    movel([0.226532, -1.331171, -2.606399, -0.774819, 1.570796, 1.797328],accel_mss,speed_ms,0,blend_radius_m)
    movel([0.225717, -1.333588, -2.604857, -0.773944, 1.570796, 1.796514],accel_mss,speed_ms,0,blend_radius_m)
    movel([0.224908, -1.335996, -2.603314, -0.773080, 1.570796, 1.795704],accel_mss,speed_ms,0,blend_radius_m)
    movel([0.224102, -1.338394, -2.601768, -0.772227, 1.570796, 1.794898],accel_mss,speed_ms,0,blend_radius_m)
    movel([0.223301, -1.340783, -2.600221, -0.771385, 1.570796, 1.794097],accel_mss,speed_ms,0,blend_radius_m)
    movel([0.222504, -1.343162, -2.598672, -0.770555, 1.570796, 1.793300],accel_mss,speed_ms,0,blend_radius_m)
    movel([0.221711, -1.345532, -2.597121, -0.769735, 1.570796, 1.792507],accel_mss,speed_ms,0,blend_radius_m)
    movel([0.220923, -1.347893, -2.595569, -0.768927, 1.570796, 1.791719],accel_mss,speed_ms,0,blend_radius_m)
    movel([0.220138, -1.350245, -2.594015, -0.768129, 1.570796, 1.790935],accel_mss,speed_ms,0,blend_radius_m)
    movel([0.219358, -1.352588, -2.592459, -0.767341, 1.570796, 1.790154],accel_mss,speed_ms,0,blend_radius_m)
    movel([0.218582, -1.354923, -2.590901, -0.766565, 1.570796, 1.789378],accel_mss,speed_ms,0,blend_radius_m)
    movel([0.217810, -1.357248, -2.589342, -0.765799, 1.570796, 1.788606],accel_mss,speed_ms,0,blend_radius_m)
    movel([0.217042, -1.359565, -2.587781, -0.765043, 1.570796, 1.787838],accel_mss,speed_ms,0,blend_radius_m)
    movel([0.216277, -1.361873, -2.586219, -0.764298, 1.570796, 1.787074],accel_mss,speed_ms,0,blend_radius_m)
    movel([0.215517, -1.364172, -2.584655, -0.763562, 1.570796, 1.786314],accel_mss,speed_ms,0,blend_radius_m)
    movel([0.214761, -1.366463, -2.583089, -0.762837, 1.570796, 1.785557],accel_mss,speed_ms,0,blend_radius_m)
    # Splitting Linear movement in 4 (instruction 613: MoveL 496)
    movel([0.212425, -1.366695, -2.582929, -0.762764, 1.570796, 1.783222],accel_mss,speed_ms,0,blend_radius_m)
    movel([0.210088, -1.366933, -2.582767, -0.762689, 1.570796, 1.780884],accel_mss,speed_ms,0,blend_radius_m)
    movel([0.207750, -1.367175, -2.582601, -0.762613, 1.570796, 1.778546],accel_mss,speed_ms,0,blend_radius_m)
    movel([0.205411, -1.367422, -2.582431, -0.762536, 1.570796, 1.776207],accel_mss,speed_ms,0,blend_radius_m)
    speed_ms = 0.003
    # Splitting Linear movement in 8 (instruction 615: MoveL 497)
    movel([0.205411, -1.365756, -2.581675, -0.764958, 1.570796, 1.776207],accel_mss,speed_ms,0,blend_radius_m)
    movel([0.205411, -1.364096, -2.580917, -0.767376, 1.570796, 1.776207],accel_mss,speed_ms,0,blend_radius_m)
    movel([0.205411, -1.362442, -2.580157, -0.769790, 1.570796, 1.776207],accel_mss,speed_ms,0,blend_radius_m)
    movel([0.205411, -1.360794, -2.579395, -0.772200, 1.570796, 1.776207],accel_mss,speed_ms,0,blend_radius_m)
    movel([0.205411, -1.359151, -2.578631, -0.774607, 1.570796, 1.776207],accel_mss,speed_ms,0,blend_radius_m)
    movel([0.205411, -1.357515, -2.577864, -0.777010, 1.570796, 1.776207],accel_mss,speed_ms,0,blend_radius_m)
    movel([0.205411, -1.355884, -2.577096, -0.779409, 1.570796, 1.776207],accel_mss,speed_ms,0,blend_radius_m)
    movel([0.205411, -1.354259, -2.576326, -0.781804, 1.570796, 1.776207],accel_mss,speed_ms,0,blend_radius_m)
    speed_ms = 1.000
    # Splitting Linear movement in 12 (instruction 617: MoveL 498)
    movel([0.205411, -1.352102, -2.575295, -0.784992, 1.570796, 1.776207],accel_mss,speed_ms,0,blend_radius_m)
    movel([0.205411, -1.349954, -2.574261, -0.788174, 1.570796, 1.776207],accel_mss,speed_ms,0,blend_radius_m)
    movel([0.205411, -1.347818, -2.573223, -0.791348, 1.570796, 1.776207],accel_mss,speed_ms,0,blend_radius_m)
    movel([0.205411, -1.345691, -2.572182, -0.794516, 1.570796, 1.776207],accel_mss,speed_ms,0,blend_radius_m)
    movel([0.205411, -1.343575, -2.571137, -0.797677, 1.570796, 1.776207],accel_mss,speed_ms,0,blend_radius_m)
    movel([0.205411, -1.341469, -2.570088, -0.800832, 1.570796, 1.776207],accel_mss,speed_ms,0,blend_radius_m)
    movel([0.205411, -1.339373, -2.569036, -0.803980, 1.570796, 1.776207],accel_mss,speed_ms,0,blend_radius_m)
    movel([0.205411, -1.337288, -2.567980, -0.807121, 1.570796, 1.776207],accel_mss,speed_ms,0,blend_radius_m)
    movel([0.205411, -1.335213, -2.566921, -0.810255, 1.570796, 1.776207],accel_mss,speed_ms,0,blend_radius_m)
    movel([0.205411, -1.333148, -2.565858, -0.813383, 1.570796, 1.776207],accel_mss,speed_ms,0,blend_radius_m)
    movel([0.205411, -1.331093, -2.564792, -0.816504, 1.570796, 1.776207],accel_mss,speed_ms,0,blend_radius_m)
    movel([0.205411, -1.329048, -2.563722, -0.819619, 1.570796, 1.776207],accel_mss,speed_ms,0,blend_radius_m)
    # Splitting Linear movement in 4 (instruction 618: MoveL 499)
    movel([0.207507, -1.328481, -2.564090, -0.819818, 1.570796, 1.778304],accel_mss,speed_ms,0,blend_radius_m)
    movel([0.209605, -1.327917, -2.564455, -0.820017, 1.570796, 1.780401],accel_mss,speed_ms,0,blend_radius_m)
    movel([0.211703, -1.327356, -2.564818, -0.820215, 1.570796, 1.782499],accel_mss,speed_ms,0,blend_radius_m)
    movel([0.213802, -1.326799, -2.565178, -0.820412, 1.570796, 1.784598],accel_mss,speed_ms,0,blend_radius_m)
    # Splitting Linear movement in 12 (instruction 619: MoveL 500)
    movel([0.213802, -1.328846, -2.566251, -0.817292, 1.570796, 1.784598],accel_mss,speed_ms,0,blend_radius_m)
    movel([0.213802, -1.330904, -2.567319, -0.814166, 1.570796, 1.784598],accel_mss,speed_ms,0,blend_radius_m)
    movel([0.213802, -1.332972, -2.568384, -0.811033, 1.570796, 1.784598],accel_mss,speed_ms,0,blend_radius_m)
    movel([0.213802, -1.335050, -2.569446, -0.807893, 1.570796, 1.784598],accel_mss,speed_ms,0,blend_radius_m)
    movel([0.213802, -1.337139, -2.570504, -0.804746, 1.570796, 1.784598],accel_mss,speed_ms,0,blend_radius_m)
    movel([0.213802, -1.339237, -2.571559, -0.801593, 1.570796, 1.784598],accel_mss,speed_ms,0,blend_radius_m)
    movel([0.213802, -1.341346, -2.572610, -0.798433, 1.570796, 1.784598],accel_mss,speed_ms,0,blend_radius_m)
    movel([0.213802, -1.343466, -2.573657, -0.795266, 1.570796, 1.784598],accel_mss,speed_ms,0,blend_radius_m)
    movel([0.213802, -1.345596, -2.574701, -0.792092, 1.570796, 1.784598],accel_mss,speed_ms,0,blend_radius_m)
    movel([0.213802, -1.347736, -2.575741, -0.788912, 1.570796, 1.784598],accel_mss,speed_ms,0,blend_radius_m)
    movel([0.213802, -1.349887, -2.576778, -0.785725, 1.570796, 1.784598],accel_mss,speed_ms,0,blend_radius_m)
    movel([0.213802, -1.352047, -2.577811, -0.782531, 1.570796, 1.784598],accel_mss,speed_ms,0,blend_radius_m)
    speed_ms = 0.003
    # Splitting Linear movement in 6 (instruction 621: MoveL 501)
    movel([0.213802, -1.353675, -2.578583, -0.780131, 1.570796, 1.784598],accel_mss,speed_ms,0,blend_radius_m)
    movel([0.213802, -1.355308, -2.579353, -0.777727, 1.570796, 1.784598],accel_mss,speed_ms,0,blend_radius_m)
    movel([0.213802, -1.356948, -2.580121, -0.775320, 1.570796, 1.784598],accel_mss,speed_ms,0,blend_radius_m)
    movel([0.213802, -1.358593, -2.580887, -0.772909, 1.570796, 1.784598],accel_mss,speed_ms,0,blend_radius_m)
    movel([0.213802, -1.360244, -2.581651, -0.770494, 1.570796, 1.784598],accel_mss,speed_ms,0,blend_radius_m)
    movel([0.213802, -1.361901, -2.582413, -0.768075, 1.570796, 1.784598],accel_mss,speed_ms,0,blend_radius_m)
    speed_ms = 0.007
    # Splitting Linear movement in 28 (instruction 623: MoveL 502)
    movel([0.214539, -1.359700, -2.583906, -0.768782, 1.570796, 1.785335],accel_mss,speed_ms,0,blend_radius_m)
    movel([0.215280, -1.357492, -2.585397, -0.769499, 1.570796, 1.786076],accel_mss,speed_ms,0,blend_radius_m)
    movel([0.216024, -1.355276, -2.586887, -0.770226, 1.570796, 1.786820],accel_mss,speed_ms,0,blend_radius_m)
    movel([0.216772, -1.353052, -2.588375, -0.770962, 1.570796, 1.787569],accel_mss,speed_ms,0,blend_radius_m)
    movel([0.217524, -1.350820, -2.589862, -0.771707, 1.570796, 1.788321],accel_mss,speed_ms,0,blend_radius_m)
    movel([0.218280, -1.348579, -2.591347, -0.772462, 1.570796, 1.789076],accel_mss,speed_ms,0,blend_radius_m)
    movel([0.219040, -1.346331, -2.592831, -0.773227, 1.570796, 1.789836],accel_mss,speed_ms,0,blend_radius_m)
    movel([0.219803, -1.344074, -2.594313, -0.774002, 1.570796, 1.790599],accel_mss,speed_ms,0,blend_radius_m)
    movel([0.220570, -1.341809, -2.595793, -0.774786, 1.570796, 1.791367],accel_mss,speed_ms,0,blend_radius_m)
    movel([0.221341, -1.339536, -2.597272, -0.775581, 1.570796, 1.792138],accel_mss,speed_ms,0,blend_radius_m)
    movel([0.222116, -1.337254, -2.598749, -0.776385, 1.570796, 1.792913],accel_mss,speed_ms,0,blend_radius_m)
    movel([0.222895, -1.334964, -2.600225, -0.777200, 1.570796, 1.793692],accel_mss,speed_ms,0,blend_radius_m)
    movel([0.223679, -1.332665, -2.601699, -0.778024, 1.570796, 1.794475],accel_mss,speed_ms,0,blend_radius_m)
    movel([0.224466, -1.330358, -2.603171, -0.778860, 1.570796, 1.795262],accel_mss,speed_ms,0,blend_radius_m)
    movel([0.225257, -1.328042, -2.604642, -0.779705, 1.570796, 1.796053],accel_mss,speed_ms,0,blend_radius_m)
    movel([0.226052, -1.325717, -2.606111, -0.780561, 1.570796, 1.796848],accel_mss,speed_ms,0,blend_radius_m)
    movel([0.226851, -1.323383, -2.607578, -0.781427, 1.570796, 1.797648],accel_mss,speed_ms,0,blend_radius_m)
    movel([0.227655, -1.321040, -2.609044, -0.782305, 1.570796, 1.798451],accel_mss,speed_ms,0,blend_radius_m)
    movel([0.228462, -1.318689, -2.610508, -0.783192, 1.570796, 1.799259],accel_mss,speed_ms,0,blend_radius_m)
    movel([0.229274, -1.316328, -2.611970, -0.784091, 1.570796, 1.800071],accel_mss,speed_ms,0,blend_radius_m)
    movel([0.230091, -1.313958, -2.613431, -0.785001, 1.570796, 1.800887],accel_mss,speed_ms,0,blend_radius_m)
    movel([0.230911, -1.311578, -2.614889, -0.785921, 1.570796, 1.801707],accel_mss,speed_ms,0,blend_radius_m)
    movel([0.231736, -1.309190, -2.616346, -0.786853, 1.570796, 1.802532],accel_mss,speed_ms,0,blend_radius_m)
    movel([0.232565, -1.306792, -2.617802, -0.787796, 1.570796, 1.803361],accel_mss,speed_ms,0,blend_radius_m)
    movel([0.233399, -1.304384, -2.619255, -0.788750, 1.570796, 1.804195],accel_mss,speed_ms,0,blend_radius_m)
    movel([0.234237, -1.301967, -2.620707, -0.789716, 1.570796, 1.805033],accel_mss,speed_ms,0,blend_radius_m)
    movel([0.235079, -1.299540, -2.622156, -0.790693, 1.570796, 1.805875],accel_mss,speed_ms,0,blend_radius_m)
    movel([0.235926, -1.297103, -2.623604, -0.791681, 1.570796, 1.806722],accel_mss,speed_ms,0,blend_radius_m)
    # Splitting Linear movement in 6 (instruction 624: MoveC 503)
    movel([0.238136, -1.297220, -2.623535, -0.791634, 1.570796, 1.808932],accel_mss,speed_ms,0,blend_radius_m)
    movel([0.240342, -1.297342, -2.623463, -0.791584, 1.570796, 1.811138],accel_mss,speed_ms,0,blend_radius_m)
    movel([0.242546, -1.297469, -2.623388, -0.791532, 1.570796, 1.813342],accel_mss,speed_ms,0,blend_radius_m)
    movel([0.244746, -1.297602, -2.623309, -0.791478, 1.570796, 1.815543],accel_mss,speed_ms,0,blend_radius_m)
    movel([0.246944, -1.297740, -2.623227, -0.791422, 1.570796, 1.817740],accel_mss,speed_ms,0,blend_radius_m)
    movel([0.249138, -1.297883, -2.623142, -0.791364, 1.570796, 1.819935],accel_mss,speed_ms,0,blend_radius_m)
    # Splitting Linear movement in 12 (instruction 625: MoveC 504)
    movel([0.250068, -1.299641, -2.622096, -0.790652, 1.570796, 1.820865],accel_mss,speed_ms,0,blend_radius_m)
    movel([0.250994, -1.301398, -2.621047, -0.789944, 1.570796, 1.821791],accel_mss,speed_ms,0,blend_radius_m)
    movel([0.251916, -1.303152, -2.619996, -0.789241, 1.570796, 1.822712],accel_mss,speed_ms,0,blend_radius_m)
    movel([0.252833, -1.304905, -2.618941, -0.788543, 1.570796, 1.823629],accel_mss,speed_ms,0,blend_radius_m)
    movel([0.253746, -1.306655, -2.617884, -0.787850, 1.570796, 1.824542],accel_mss,speed_ms,0,blend_radius_m)
    movel([0.254655, -1.308403, -2.616824, -0.787161, 1.570796, 1.825451],accel_mss,speed_ms,0,blend_radius_m)
    movel([0.255560, -1.310150, -2.615762, -0.786478, 1.570796, 1.826356],accel_mss,speed_ms,0,blend_radius_m)
    movel([0.256461, -1.311894, -2.614696, -0.785799, 1.570796, 1.827257],accel_mss,speed_ms,0,blend_radius_m)
    movel([0.257357, -1.313636, -2.613628, -0.785125, 1.570796, 1.828154],accel_mss,speed_ms,0,blend_radius_m)
    movel([0.258250, -1.315377, -2.612557, -0.784455, 1.570796, 1.829046],accel_mss,speed_ms,0,blend_radius_m)
    movel([0.259138, -1.317115, -2.611484, -0.783791, 1.570796, 1.829934],accel_mss,speed_ms,0,blend_radius_m)
    movel([0.260023, -1.318851, -2.610407, -0.783131, 1.570796, 1.830819],accel_mss,speed_ms,0,blend_radius_m)
    movel([0.259481, -1.321910, -2.608501, -0.781978, 1.570796, 1.830277],accel_mss,speed_ms,0,blend_radius_m)
    movel([0.259060, -1.323596, -2.607445, -0.781348, 1.570796, 1.829856],accel_mss,speed_ms,0,blend_radius_m)
    movel([0.258139, -1.326541, -2.605592, -0.780257, 1.570796, 1.828935],accel_mss,speed_ms,0,blend_radius_m)
    movel([0.256608, -1.330373, -2.603162, -0.778854, 1.570796, 1.827405],accel_mss,speed_ms,0,blend_radius_m)
    movel([0.255647, -1.332392, -2.601874, -0.778123, 1.570796, 1.826443],accel_mss,speed_ms,0,blend_radius_m)
    movel([0.254869, -1.333870, -2.600928, -0.777592, 1.570796, 1.825665],accel_mss,speed_ms,0,blend_radius_m)
    # Splitting Linear movement in 8 (instruction 632: MoveC 511)
    movel([0.253270, -1.335839, -2.599662, -0.776888, 1.570796, 1.824066],accel_mss,speed_ms,0,blend_radius_m)
    movel([0.251678, -1.337802, -2.598395, -0.776191, 1.570796, 1.822474],accel_mss,speed_ms,0,blend_radius_m)
    movel([0.250091, -1.339760, -2.597127, -0.775502, 1.570796, 1.820888],accel_mss,speed_ms,0,blend_radius_m)
    movel([0.248511, -1.341712, -2.595857, -0.774820, 1.570796, 1.819308],accel_mss,speed_ms,0,blend_radius_m)
    movel([0.246938, -1.343658, -2.594586, -0.774145, 1.570796, 1.817734],accel_mss,speed_ms,0,blend_radius_m)
    movel([0.245370, -1.345598, -2.593313, -0.773478, 1.570796, 1.816166],accel_mss,speed_ms,0,blend_radius_m)
    movel([0.243809, -1.347533, -2.592038, -0.772817, 1.570796, 1.814605],accel_mss,speed_ms,0,blend_radius_m)
    movel([0.242253, -1.349462, -2.590763, -0.772164, 1.570796, 1.813050],accel_mss,speed_ms,0,blend_radius_m)
    # Splitting Linear movement in 4 (instruction 633: MoveC 512)
    movel([0.240979, -1.350466, -2.590097, -0.771826, 1.570796, 1.811775],accel_mss,speed_ms,0,blend_radius_m)
    movel([0.239707, -1.351470, -2.589430, -0.771489, 1.570796, 1.810503],accel_mss,speed_ms,0,blend_radius_m)
    movel([0.238437, -1.352472, -2.588763, -0.771155, 1.570796, 1.809234],accel_mss,speed_ms,0,blend_radius_m)
    movel([0.237170, -1.353473, -2.588094, -0.770822, 1.570796, 1.807966],accel_mss,speed_ms,0,blend_radius_m)
    movel([0.235144, -1.354822, -2.587191, -0.770375, 1.570796, 1.805940],accel_mss,speed_ms,0,blend_radius_m)
    # Splitting Linear movement in 8 (instruction 635: MoveC 514)
    movel([0.233110, -1.355638, -2.586644, -0.770107, 1.570796, 1.803906],accel_mss,speed_ms,0,blend_radius_m)
    movel([0.231078, -1.356455, -2.586095, -0.769838, 1.570796, 1.801874],accel_mss,speed_ms,0,blend_radius_m)
    movel([0.229048, -1.357274, -2.585544, -0.769571, 1.570796, 1.799845],accel_mss,speed_ms,0,blend_radius_m)
    movel([0.227021, -1.358095, -2.584991, -0.769303, 1.570796, 1.797817],accel_mss,speed_ms,0,blend_radius_m)
    movel([0.224995, -1.358917, -2.584436, -0.769036, 1.570796, 1.795791],accel_mss,speed_ms,0,blend_radius_m)
    movel([0.222972, -1.359741, -2.583878, -0.768769, 1.570796, 1.793768],accel_mss,speed_ms,0,blend_radius_m)
    movel([0.220950, -1.360567, -2.583319, -0.768503, 1.570796, 1.791747],accel_mss,speed_ms,0,blend_radius_m)
    movel([0.218931, -1.361394, -2.582758, -0.768237, 1.570796, 1.789728],accel_mss,speed_ms,0,blend_radius_m)
    # Splitting Linear movement in 4 (instruction 636: MoveC 515)
    movel([0.217650, -1.361519, -2.582673, -0.768197, 1.570796, 1.788446],accel_mss,speed_ms,0,blend_radius_m)
    movel([0.216367, -1.361645, -2.582587, -0.768157, 1.570796, 1.787164],accel_mss,speed_ms,0,blend_radius_m)
    movel([0.215085, -1.361772, -2.582501, -0.768116, 1.570796, 1.785881],accel_mss,speed_ms,0,blend_radius_m)
    movel([0.213802, -1.361901, -2.582413, -0.768075, 1.570796, 1.784598],accel_mss,speed_ms,0,blend_radius_m)
    speed_ms = 0.003
    movel([0.213802, -1.365233, -2.583931, -0.763226, 1.570796, 1.784598],accel_mss,speed_ms,0,blend_radius_m)
    speed_ms = 0.007
    # Splitting Linear movement in 28 (instruction 640: MoveL 517)
    movel([0.214539, -1.363038, -2.585427, -0.763924, 1.570796, 1.785335],accel_mss,speed_ms,0,blend_radius_m)
    movel([0.215280, -1.360835, -2.586922, -0.764632, 1.570796, 1.786076],accel_mss,speed_ms,0,blend_radius_m)
    movel([0.216024, -1.358625, -2.588416, -0.765349, 1.570796, 1.786820],accel_mss,speed_ms,0,blend_radius_m)
    movel([0.216772, -1.356406, -2.589908, -0.766075, 1.570796, 1.787569],accel_mss,speed_ms,0,blend_radius_m)
    movel([0.217524, -1.354180, -2.591398, -0.766811, 1.570796, 1.788321],accel_mss,speed_ms,0,blend_radius_m)
    movel([0.218280, -1.351945, -2.592887, -0.767557, 1.570796, 1.789076],accel_mss,speed_ms,0,blend_radius_m)
    movel([0.219040, -1.349703, -2.594374, -0.768312, 1.570796, 1.789836],accel_mss,speed_ms,0,blend_radius_m)
    movel([0.219803, -1.347452, -2.595860, -0.769077, 1.570796, 1.790599],accel_mss,speed_ms,0,blend_radius_m)
    movel([0.220570, -1.345192, -2.597344, -0.769852, 1.570796, 1.791367],accel_mss,speed_ms,0,blend_radius_m)
    movel([0.221341, -1.342925, -2.598827, -0.770637, 1.570796, 1.792138],accel_mss,speed_ms,0,blend_radius_m)
    movel([0.222116, -1.340649, -2.600308, -0.771432, 1.570796, 1.792913],accel_mss,speed_ms,0,blend_radius_m)
    movel([0.222895, -1.338364, -2.601787, -0.772237, 1.570796, 1.793692],accel_mss,speed_ms,0,blend_radius_m)
    movel([0.223679, -1.336071, -2.603265, -0.773053, 1.570796, 1.794475],accel_mss,speed_ms,0,blend_radius_m)
    movel([0.224466, -1.333769, -2.604741, -0.773878, 1.570796, 1.795262],accel_mss,speed_ms,0,blend_radius_m)
    movel([0.225257, -1.331459, -2.606216, -0.774714, 1.570796, 1.796053],accel_mss,speed_ms,0,blend_radius_m)
    movel([0.226052, -1.329140, -2.607689, -0.775561, 1.570796, 1.796848],accel_mss,speed_ms,0,blend_radius_m)
    movel([0.226851, -1.326811, -2.609160, -0.776418, 1.570796, 1.797648],accel_mss,speed_ms,0,blend_radius_m)
    movel([0.227655, -1.324474, -2.610630, -0.777285, 1.570796, 1.798451],accel_mss,speed_ms,0,blend_radius_m)
    movel([0.228462, -1.322128, -2.612098, -0.778163, 1.570796, 1.799259],accel_mss,speed_ms,0,blend_radius_m)
    movel([0.229274, -1.319773, -2.613564, -0.779053, 1.570796, 1.800071],accel_mss,speed_ms,0,blend_radius_m)
    movel([0.230091, -1.317408, -2.615028, -0.779953, 1.570796, 1.800887],accel_mss,speed_ms,0,blend_radius_m)
    movel([0.230911, -1.315034, -2.616491, -0.780864, 1.570796, 1.801707],accel_mss,speed_ms,0,blend_radius_m)
    movel([0.231736, -1.312651, -2.617952, -0.781786, 1.570796, 1.802532],accel_mss,speed_ms,0,blend_radius_m)
    movel([0.232565, -1.310259, -2.619411, -0.782719, 1.570796, 1.803361],accel_mss,speed_ms,0,blend_radius_m)
    movel([0.233399, -1.307857, -2.620869, -0.783664, 1.570796, 1.804195],accel_mss,speed_ms,0,blend_radius_m)
    movel([0.234237, -1.305445, -2.622325, -0.784620, 1.570796, 1.805033],accel_mss,speed_ms,0,blend_radius_m)
    movel([0.235079, -1.303023, -2.623778, -0.785587, 1.570796, 1.805875],accel_mss,speed_ms,0,blend_radius_m)
    movel([0.235926, -1.300592, -2.625231, -0.786566, 1.570796, 1.806722],accel_mss,speed_ms,0,blend_radius_m)
    # Splitting Linear movement in 6 (instruction 641: MoveC 518)
    movel([0.238136, -1.300709, -2.625161, -0.786519, 1.570796, 1.808932],accel_mss,speed_ms,0,blend_radius_m)
    movel([0.240342, -1.300830, -2.625089, -0.786470, 1.570796, 1.811138],accel_mss,speed_ms,0,blend_radius_m)
    movel([0.242546, -1.300957, -2.625013, -0.786419, 1.570796, 1.813342],accel_mss,speed_ms,0,blend_radius_m)
    movel([0.244746, -1.301090, -2.624934, -0.786365, 1.570796, 1.815543],accel_mss,speed_ms,0,blend_radius_m)
    movel([0.246944, -1.301227, -2.624852, -0.786310, 1.570796, 1.817740],accel_mss,speed_ms,0,blend_radius_m)
    movel([0.249138, -1.301370, -2.624767, -0.786252, 1.570796, 1.819935],accel_mss,speed_ms,0,blend_radius_m)
    # Splitting Linear movement in 12 (instruction 642: MoveC 519)
    movel([0.250068, -1.303125, -2.623718, -0.785547, 1.570796, 1.820865],accel_mss,speed_ms,0,blend_radius_m)
    movel([0.250994, -1.304877, -2.622666, -0.784846, 1.570796, 1.821791],accel_mss,speed_ms,0,blend_radius_m)
    movel([0.251916, -1.306628, -2.621612, -0.784150, 1.570796, 1.822712],accel_mss,speed_ms,0,blend_radius_m)
    movel([0.252833, -1.308376, -2.620554, -0.783459, 1.570796, 1.823629],accel_mss,speed_ms,0,blend_radius_m)
    movel([0.253746, -1.310122, -2.619494, -0.782772, 1.570796, 1.824542],accel_mss,speed_ms,0,blend_radius_m)
    movel([0.254655, -1.311867, -2.618431, -0.782091, 1.570796, 1.825451],accel_mss,speed_ms,0,blend_radius_m)
    movel([0.255560, -1.313609, -2.617366, -0.781414, 1.570796, 1.826356],accel_mss,speed_ms,0,blend_radius_m)
    movel([0.256461, -1.315349, -2.616297, -0.780742, 1.570796, 1.827257],accel_mss,speed_ms,0,blend_radius_m)
    movel([0.257357, -1.317088, -2.615226, -0.780075, 1.570796, 1.828154],accel_mss,speed_ms,0,blend_radius_m)
    movel([0.258250, -1.318824, -2.614152, -0.779413, 1.570796, 1.829046],accel_mss,speed_ms,0,blend_radius_m)
    movel([0.259138, -1.320558, -2.613076, -0.778755, 1.570796, 1.829934],accel_mss,speed_ms,0,blend_radius_m)
    movel([0.260023, -1.322290, -2.611997, -0.778103, 1.570796, 1.830819],accel_mss,speed_ms,0,blend_radius_m)
    movel([0.259481, -1.325342, -2.610085, -0.776962, 1.570796, 1.830277],accel_mss,speed_ms,0,blend_radius_m)
    movel([0.259060, -1.327024, -2.609026, -0.776339, 1.570796, 1.829856],accel_mss,speed_ms,0,blend_radius_m)
    movel([0.258139, -1.329961, -2.607168, -0.775260, 1.570796, 1.828935],accel_mss,speed_ms,0,blend_radius_m)
    movel([0.256608, -1.333784, -2.604732, -0.773873, 1.570796, 1.827405],accel_mss,speed_ms,0,blend_radius_m)
    movel([0.255647, -1.335798, -2.603441, -0.773150, 1.570796, 1.826443],accel_mss,speed_ms,0,blend_radius_m)
    movel([0.254869, -1.337272, -2.602492, -0.772625, 1.570796, 1.825665],accel_mss,speed_ms,0,blend_radius_m)
    # Splitting Linear movement in 8 (instruction 649: MoveC 526)
    movel([0.253270, -1.339237, -2.601223, -0.771929, 1.570796, 1.824066],accel_mss,speed_ms,0,blend_radius_m)
    movel([0.251678, -1.341195, -2.599953, -0.771241, 1.570796, 1.822474],accel_mss,speed_ms,0,blend_radius_m)
    movel([0.250091, -1.343148, -2.598681, -0.770560, 1.570796, 1.820888],accel_mss,speed_ms,0,blend_radius_m)
    movel([0.248511, -1.345095, -2.597408, -0.769886, 1.570796, 1.819308],accel_mss,speed_ms,0,blend_radius_m)
    movel([0.246938, -1.347036, -2.596133, -0.769219, 1.570796, 1.817734],accel_mss,speed_ms,0,blend_radius_m)
    movel([0.245370, -1.348972, -2.594857, -0.768560, 1.570796, 1.816166],accel_mss,speed_ms,0,blend_radius_m)
    movel([0.243809, -1.350902, -2.593580, -0.767907, 1.570796, 1.814605],accel_mss,speed_ms,0,blend_radius_m)
    movel([0.242253, -1.352826, -2.592301, -0.767262, 1.570796, 1.813050],accel_mss,speed_ms,0,blend_radius_m)
    # Splitting Linear movement in 4 (instruction 650: MoveC 527)
    movel([0.240979, -1.353828, -2.591633, -0.766928, 1.570796, 1.811775],accel_mss,speed_ms,0,blend_radius_m)
    movel([0.239707, -1.354828, -2.590965, -0.766596, 1.570796, 1.810503],accel_mss,speed_ms,0,blend_radius_m)
    movel([0.238437, -1.355828, -2.590296, -0.766266, 1.570796, 1.809234],accel_mss,speed_ms,0,blend_radius_m)
    movel([0.237170, -1.356826, -2.589626, -0.765937, 1.570796, 1.807966],accel_mss,speed_ms,0,blend_radius_m)
    movel([0.235144, -1.358172, -2.588720, -0.765496, 1.570796, 1.805940],accel_mss,speed_ms,0,blend_radius_m)
    # Splitting Linear movement in 8 (instruction 652: MoveC 529)
    movel([0.233110, -1.358986, -2.588172, -0.765231, 1.570796, 1.803906],accel_mss,speed_ms,0,blend_radius_m)
    movel([0.231078, -1.359801, -2.587622, -0.764966, 1.570796, 1.801874],accel_mss,speed_ms,0,blend_radius_m)
    movel([0.229048, -1.360618, -2.587069, -0.764702, 1.570796, 1.799845],accel_mss,speed_ms,0,blend_radius_m)
    movel([0.227021, -1.361436, -2.586515, -0.764438, 1.570796, 1.797817],accel_mss,speed_ms,0,blend_radius_m)
    movel([0.224995, -1.362257, -2.585958, -0.764174, 1.570796, 1.795791],accel_mss,speed_ms,0,blend_radius_m)
    movel([0.222972, -1.363079, -2.585399, -0.763911, 1.570796, 1.793768],accel_mss,speed_ms,0,blend_radius_m)
    movel([0.220950, -1.363902, -2.584839, -0.763648, 1.570796, 1.791747],accel_mss,speed_ms,0,blend_radius_m)
    movel([0.218931, -1.364727, -2.584276, -0.763386, 1.570796, 1.789728],accel_mss,speed_ms,0,blend_radius_m)
    # Splitting Linear movement in 4 (instruction 653: MoveC 530)
    movel([0.217650, -1.364851, -2.584191, -0.763347, 1.570796, 1.788446],accel_mss,speed_ms,0,blend_radius_m)
    movel([0.216367, -1.364977, -2.584105, -0.763307, 1.570796, 1.787164],accel_mss,speed_ms,0,blend_radius_m)
    movel([0.215085, -1.365104, -2.584018, -0.763266, 1.570796, 1.785881],accel_mss,speed_ms,0,blend_radius_m)
    movel([0.213802, -1.365233, -2.583931, -0.763226, 1.570796, 1.784598],accel_mss,speed_ms,0,blend_radius_m)
    speed_ms = 0.003
    # Splitting Linear movement in 6 (instruction 655: MoveL 531)
    movel([0.213802, -1.363009, -2.582920, -0.766460, 1.570796, 1.784598],accel_mss,speed_ms,0,blend_radius_m)
    movel([0.213802, -1.360796, -2.581906, -0.769688, 1.570796, 1.784598],accel_mss,speed_ms,0,blend_radius_m)
    movel([0.213802, -1.358593, -2.580887, -0.772909, 1.570796, 1.784598],accel_mss,speed_ms,0,blend_radius_m)
    movel([0.213802, -1.356401, -2.579865, -0.776123, 1.570796, 1.784598],accel_mss,speed_ms,0,blend_radius_m)
    movel([0.213802, -1.354219, -2.578840, -0.779330, 1.570796, 1.784598],accel_mss,speed_ms,0,blend_radius_m)
    movel([0.213802, -1.352047, -2.577811, -0.782531, 1.570796, 1.784598],accel_mss,speed_ms,0,blend_radius_m)
    speed_ms = 1.000
    # Splitting Linear movement in 12 (instruction 657: MoveL 532)
    movel([0.213802, -1.349887, -2.576778, -0.785725, 1.570796, 1.784598],accel_mss,speed_ms,0,blend_radius_m)
    movel([0.213802, -1.347736, -2.575741, -0.788912, 1.570796, 1.784598],accel_mss,speed_ms,0,blend_radius_m)
    movel([0.213802, -1.345596, -2.574701, -0.792092, 1.570796, 1.784598],accel_mss,speed_ms,0,blend_radius_m)
    movel([0.213802, -1.343466, -2.573657, -0.795266, 1.570796, 1.784598],accel_mss,speed_ms,0,blend_radius_m)
    movel([0.213802, -1.341346, -2.572610, -0.798433, 1.570796, 1.784598],accel_mss,speed_ms,0,blend_radius_m)
    movel([0.213802, -1.339237, -2.571559, -0.801593, 1.570796, 1.784598],accel_mss,speed_ms,0,blend_radius_m)
    movel([0.213802, -1.337139, -2.570504, -0.804746, 1.570796, 1.784598],accel_mss,speed_ms,0,blend_radius_m)
    movel([0.213802, -1.335050, -2.569446, -0.807893, 1.570796, 1.784598],accel_mss,speed_ms,0,blend_radius_m)
    movel([0.213802, -1.332972, -2.568384, -0.811033, 1.570796, 1.784598],accel_mss,speed_ms,0,blend_radius_m)
    movel([0.213802, -1.330904, -2.567319, -0.814166, 1.570796, 1.784598],accel_mss,speed_ms,0,blend_radius_m)
    movel([0.213802, -1.328846, -2.566251, -0.817292, 1.570796, 1.784598],accel_mss,speed_ms,0,blend_radius_m)
    movel([0.213802, -1.326799, -2.565178, -0.820412, 1.570796, 1.784598],accel_mss,speed_ms,0,blend_radius_m)
    # Splitting Linear movement in 18 (instruction 658: MoveL 533)
    movel([0.215158, -1.324599, -2.566596, -0.821194, 1.570796, 1.785954],accel_mss,speed_ms,0,blend_radius_m)
    movel([0.216520, -1.322393, -2.568011, -0.821985, 1.570796, 1.787317],accel_mss,speed_ms,0,blend_radius_m)
    movel([0.217889, -1.320180, -2.569425, -0.822785, 1.570796, 1.788685],accel_mss,speed_ms,0,blend_radius_m)
    movel([0.219264, -1.317959, -2.570837, -0.823593, 1.570796, 1.790060],accel_mss,speed_ms,0,blend_radius_m)
    movel([0.220645, -1.315730, -2.572247, -0.824411, 1.570796, 1.791441],accel_mss,speed_ms,0,blend_radius_m)
    movel([0.222033, -1.313495, -2.573656, -0.825238, 1.570796, 1.792829],accel_mss,speed_ms,0,blend_radius_m)
    movel([0.223426, -1.311251, -2.575063, -0.826075, 1.570796, 1.794223],accel_mss,speed_ms,0,blend_radius_m)
    movel([0.224827, -1.309001, -2.576468, -0.826920, 1.570796, 1.795623],accel_mss,speed_ms,0,blend_radius_m)
    movel([0.226234, -1.306742, -2.577872, -0.827775, 1.570796, 1.797030],accel_mss,speed_ms,0,blend_radius_m)
    movel([0.227647, -1.304476, -2.579273, -0.828640, 1.570796, 1.798444],accel_mss,speed_ms,0,blend_radius_m)
    movel([0.229067, -1.302202, -2.580673, -0.829513, 1.570796, 1.799864],accel_mss,speed_ms,0,blend_radius_m)
    movel([0.230494, -1.299921, -2.582071, -0.830397, 1.570796, 1.801290],accel_mss,speed_ms,0,blend_radius_m)
    movel([0.231927, -1.297632, -2.583468, -0.831290, 1.570796, 1.802724],accel_mss,speed_ms,0,blend_radius_m)
    movel([0.233367, -1.295334, -2.584862, -0.832193, 1.570796, 1.804164],accel_mss,speed_ms,0,blend_radius_m)
    movel([0.234814, -1.293029, -2.586255, -0.833105, 1.570796, 1.805610],accel_mss,speed_ms,0,blend_radius_m)
    movel([0.236268, -1.290716, -2.587646, -0.834028, 1.570796, 1.807064],accel_mss,speed_ms,0,blend_radius_m)
    movel([0.237728, -1.288394, -2.589035, -0.834960, 1.570796, 1.808525],accel_mss,speed_ms,0,blend_radius_m)
    movel([0.239196, -1.286065, -2.590422, -0.835902, 1.570796, 1.809992],accel_mss,speed_ms,0,blend_radius_m)
    # Splitting Linear movement in 12 (instruction 659: MoveL 534)
    movel([0.239196, -1.288161, -2.591538, -0.832691, 1.570796, 1.809992],accel_mss,speed_ms,0,blend_radius_m)
    movel([0.239196, -1.290267, -2.592650, -0.829471, 1.570796, 1.809992],accel_mss,speed_ms,0,blend_radius_m)
    movel([0.239196, -1.292386, -2.593759, -0.826244, 1.570796, 1.809992],accel_mss,speed_ms,0,blend_radius_m)
    movel([0.239196, -1.294515, -2.594865, -0.823009, 1.570796, 1.809992],accel_mss,speed_ms,0,blend_radius_m)
    movel([0.239196, -1.296656, -2.595967, -0.819766, 1.570796, 1.809992],accel_mss,speed_ms,0,blend_radius_m)
    movel([0.239196, -1.298808, -2.597065, -0.816516, 1.570796, 1.809992],accel_mss,speed_ms,0,blend_radius_m)
    movel([0.239196, -1.300972, -2.598160, -0.813257, 1.570796, 1.809992],accel_mss,speed_ms,0,blend_radius_m)
    movel([0.239196, -1.303147, -2.599252, -0.809991, 1.570796, 1.809992],accel_mss,speed_ms,0,blend_radius_m)
    movel([0.239196, -1.305333, -2.600340, -0.806716, 1.570796, 1.809992],accel_mss,speed_ms,0,blend_radius_m)
    movel([0.239196, -1.307531, -2.601424, -0.803434, 1.570796, 1.809992],accel_mss,speed_ms,0,blend_radius_m)
    movel([0.239196, -1.309740, -2.602505, -0.800144, 1.570796, 1.809992],accel_mss,speed_ms,0,blend_radius_m)
    movel([0.239196, -1.311961, -2.603582, -0.796846, 1.570796, 1.809992],accel_mss,speed_ms,0,blend_radius_m)
    speed_ms = 0.003
    # Splitting Linear movement in 6 (instruction 661: MoveL 535)
    movel([0.239196, -1.313634, -2.604387, -0.794368, 1.570796, 1.809992],accel_mss,speed_ms,0,blend_radius_m)
    movel([0.239196, -1.315314, -2.605191, -0.791884, 1.570796, 1.809992],accel_mss,speed_ms,0,blend_radius_m)
    movel([0.239196, -1.317000, -2.605992, -0.789397, 1.570796, 1.809992],accel_mss,speed_ms,0,blend_radius_m)
    movel([0.239196, -1.318693, -2.606791, -0.786905, 1.570796, 1.809992],accel_mss,speed_ms,0,blend_radius_m)
    movel([0.239196, -1.320392, -2.607588, -0.784409, 1.570796, 1.809992],accel_mss,speed_ms,0,blend_radius_m)
    movel([0.239196, -1.322098, -2.608383, -0.781908, 1.570796, 1.809992],accel_mss,speed_ms,0,blend_radius_m)
    speed_ms = 0.007
    # Splitting Linear movement in 4 (instruction 663: MoveC 536)
    movel([0.238117, -1.321461, -2.608781, -0.782146, 1.570796, 1.808913],accel_mss,speed_ms,0,blend_radius_m)
    movel([0.237036, -1.320826, -2.609178, -0.782385, 1.570796, 1.807833],accel_mss,speed_ms,0,blend_radius_m)
    movel([0.235953, -1.320192, -2.609573, -0.782624, 1.570796, 1.806750],accel_mss,speed_ms,0,blend_radius_m)
    movel([0.234868, -1.319559, -2.609967, -0.782863, 1.570796, 1.805664],accel_mss,speed_ms,0,blend_radius_m)
    movel([0.235037, -1.314955, -2.612817, -0.784617, 1.570796, 1.805833],accel_mss,speed_ms,0,blend_radius_m)
    # Splitting Linear movement in 4 (instruction 665: MoveC 538)
    movel([0.235966, -1.313583, -2.613661, -0.785145, 1.570796, 1.806762],accel_mss,speed_ms,0,blend_radius_m)
    movel([0.236897, -1.312208, -2.614504, -0.785677, 1.570796, 1.807694],accel_mss,speed_ms,0,blend_radius_m)
    movel([0.237832, -1.310830, -2.615347, -0.786212, 1.570796, 1.808628],accel_mss,speed_ms,0,blend_radius_m)
    movel([0.238769, -1.309448, -2.616189, -0.786752, 1.570796, 1.809565],accel_mss,speed_ms,0,blend_radius_m)
    # Splitting Linear movement in 4 (instruction 666: MoveC 539)
    movel([0.240367, -1.308658, -2.616670, -0.787061, 1.570796, 1.811164],accel_mss,speed_ms,0,blend_radius_m)
    movel([0.241968, -1.307867, -2.617150, -0.787372, 1.570796, 1.812764],accel_mss,speed_ms,0,blend_radius_m)
    movel([0.243570, -1.307078, -2.617628, -0.787683, 1.570796, 1.814366],accel_mss,speed_ms,0,blend_radius_m)
    movel([0.245174, -1.306289, -2.618106, -0.787995, 1.570796, 1.815970],accel_mss,speed_ms,0,blend_radius_m)
    movel([0.245654, -1.306259, -2.618124, -0.788006, 1.570796, 1.816450],accel_mss,speed_ms,0,blend_radius_m)
    # Splitting Linear movement in 4 (instruction 668: MoveC 541)
    movel([0.246742, -1.306911, -2.617729, -0.787749, 1.570796, 1.817539],accel_mss,speed_ms,0,blend_radius_m)
    movel([0.247828, -1.307565, -2.617333, -0.787491, 1.570796, 1.818625],accel_mss,speed_ms,0,blend_radius_m)
    movel([0.248912, -1.308220, -2.616936, -0.787233, 1.570796, 1.819708],accel_mss,speed_ms,0,blend_radius_m)
    movel([0.249994, -1.308876, -2.616537, -0.786976, 1.570796, 1.820790],accel_mss,speed_ms,0,blend_radius_m)
    movel([0.249744, -1.313555, -2.613678, -0.785156, 1.570796, 1.820541],accel_mss,speed_ms,0,blend_radius_m)
    # Splitting Linear movement in 4 (instruction 670: MoveC 543)
    movel([0.248800, -1.314923, -2.612837, -0.784629, 1.570796, 1.819596],accel_mss,speed_ms,0,blend_radius_m)
    movel([0.247858, -1.316287, -2.611996, -0.784107, 1.570796, 1.818654],accel_mss,speed_ms,0,blend_radius_m)
    movel([0.246918, -1.317648, -2.611154, -0.783588, 1.570796, 1.817715],accel_mss,speed_ms,0,blend_radius_m)
    movel([0.245982, -1.319006, -2.610311, -0.783072, 1.570796, 1.816778],accel_mss,speed_ms,0,blend_radius_m)
    # Splitting Linear movement in 4 (instruction 671: MoveC 544)
    movel([0.244401, -1.319771, -2.609835, -0.782783, 1.570796, 1.815197],accel_mss,speed_ms,0,blend_radius_m)
    movel([0.242822, -1.320536, -2.609358, -0.782494, 1.570796, 1.813618],accel_mss,speed_ms,0,blend_radius_m)
    movel([0.241244, -1.321303, -2.608880, -0.782206, 1.570796, 1.812040],accel_mss,speed_ms,0,blend_radius_m)
    movel([0.239668, -1.322069, -2.608401, -0.781918, 1.570796, 1.810464],accel_mss,speed_ms,0,blend_radius_m)
    movel([0.239196, -1.322098, -2.608383, -0.781908, 1.570796, 1.809992],accel_mss,speed_ms,0,blend_radius_m)
    speed_ms = 0.003
    movel([0.239196, -1.325529, -2.609967, -0.776893, 1.570796, 1.809992],accel_mss,speed_ms,0,blend_radius_m)
    speed_ms = 0.007
    # Splitting Linear movement in 4 (instruction 676: MoveC 547)
    movel([0.238117, -1.324894, -2.610366, -0.777129, 1.570796, 1.808913],accel_mss,speed_ms,0,blend_radius_m)
    movel([0.237036, -1.324260, -2.610764, -0.777365, 1.570796, 1.807833],accel_mss,speed_ms,0,blend_radius_m)
    movel([0.235953, -1.323628, -2.611160, -0.777601, 1.570796, 1.806750],accel_mss,speed_ms,0,blend_radius_m)
    movel([0.234868, -1.322997, -2.611555, -0.777837, 1.570796, 1.805664],accel_mss,speed_ms,0,blend_radius_m)
    movel([0.235037, -1.318403, -2.614413, -0.779573, 1.570796, 1.805833],accel_mss,speed_ms,0,blend_radius_m)
    # Splitting Linear movement in 4 (instruction 678: MoveC 549)
    movel([0.235966, -1.317034, -2.615259, -0.780096, 1.570796, 1.806762],accel_mss,speed_ms,0,blend_radius_m)
    movel([0.236897, -1.315662, -2.616105, -0.780622, 1.570796, 1.807694],accel_mss,speed_ms,0,blend_radius_m)
    movel([0.237832, -1.314287, -2.616950, -0.781152, 1.570796, 1.808628],accel_mss,speed_ms,0,blend_radius_m)
    movel([0.238769, -1.312909, -2.617794, -0.781686, 1.570796, 1.809565],accel_mss,speed_ms,0,blend_radius_m)
    # Splitting Linear movement in 4 (instruction 679: MoveC 550)
    movel([0.240367, -1.312120, -2.618276, -0.781992, 1.570796, 1.811164],accel_mss,speed_ms,0,blend_radius_m)
    movel([0.241968, -1.311332, -2.618758, -0.782299, 1.570796, 1.812764],accel_mss,speed_ms,0,blend_radius_m)
    movel([0.243570, -1.310544, -2.619238, -0.782607, 1.570796, 1.814366],accel_mss,speed_ms,0,blend_radius_m)
    movel([0.245174, -1.309757, -2.619716, -0.782916, 1.570796, 1.815970],accel_mss,speed_ms,0,blend_radius_m)
    movel([0.245654, -1.309727, -2.619735, -0.782928, 1.570796, 1.816450],accel_mss,speed_ms,0,blend_radius_m)
    # Splitting Linear movement in 4 (instruction 681: MoveC 552)
    movel([0.246742, -1.310378, -2.619339, -0.782672, 1.570796, 1.817539],accel_mss,speed_ms,0,blend_radius_m)
    movel([0.247828, -1.311030, -2.618942, -0.782417, 1.570796, 1.818625],accel_mss,speed_ms,0,blend_radius_m)
    movel([0.248912, -1.311684, -2.618543, -0.782162, 1.570796, 1.819708],accel_mss,speed_ms,0,blend_radius_m)
    movel([0.249994, -1.312338, -2.618143, -0.781907, 1.570796, 1.820790],accel_mss,speed_ms,0,blend_radius_m)
    movel([0.249744, -1.317007, -2.615276, -0.780106, 1.570796, 1.820541],accel_mss,speed_ms,0,blend_radius_m)
    # Splitting Linear movement in 4 (instruction 683: MoveC 554)
    movel([0.248800, -1.318371, -2.614433, -0.779585, 1.570796, 1.819596],accel_mss,speed_ms,0,blend_radius_m)
    movel([0.247858, -1.319732, -2.613589, -0.779068, 1.570796, 1.818654],accel_mss,speed_ms,0,blend_radius_m)
    movel([0.246918, -1.321090, -2.612745, -0.778555, 1.570796, 1.817715],accel_mss,speed_ms,0,blend_radius_m)
    movel([0.245982, -1.322444, -2.611900, -0.778045, 1.570796, 1.816778],accel_mss,speed_ms,0,blend_radius_m)
    # Splitting Linear movement in 4 (instruction 684: MoveC 555)
    movel([0.244401, -1.323208, -2.611423, -0.777758, 1.570796, 1.815197],accel_mss,speed_ms,0,blend_radius_m)
    movel([0.242822, -1.323971, -2.610945, -0.777473, 1.570796, 1.813618],accel_mss,speed_ms,0,blend_radius_m)
    movel([0.241244, -1.324736, -2.610466, -0.777188, 1.570796, 1.812040],accel_mss,speed_ms,0,blend_radius_m)
    movel([0.239668, -1.325501, -2.609985, -0.776903, 1.570796, 1.810464],accel_mss,speed_ms,0,blend_radius_m)
    movel([0.239196, -1.325529, -2.609967, -0.776893, 1.570796, 1.809992],accel_mss,speed_ms,0,blend_radius_m)
    speed_ms = 0.003
    # Splitting Linear movement in 6 (instruction 687: MoveL 557)
    movel([0.239196, -1.323239, -2.608912, -0.780238, 1.570796, 1.809992],accel_mss,speed_ms,0,blend_radius_m)
    movel([0.239196, -1.320960, -2.607854, -0.783575, 1.570796, 1.809992],accel_mss,speed_ms,0,blend_radius_m)
    movel([0.239196, -1.318693, -2.606791, -0.786905, 1.570796, 1.809992],accel_mss,speed_ms,0,blend_radius_m)
    movel([0.239196, -1.316437, -2.605725, -0.790227, 1.570796, 1.809992],accel_mss,speed_ms,0,blend_radius_m)
    movel([0.239196, -1.314193, -2.604655, -0.793540, 1.570796, 1.809992],accel_mss,speed_ms,0,blend_radius_m)
    movel([0.239196, -1.311961, -2.603582, -0.796846, 1.570796, 1.809992],accel_mss,speed_ms,0,blend_radius_m)
    speed_ms = 1.000
    # Splitting Linear movement in 12 (instruction 689: MoveL 558)
    movel([0.239196, -1.309740, -2.602505, -0.800144, 1.570796, 1.809992],accel_mss,speed_ms,0,blend_radius_m)
    movel([0.239196, -1.307531, -2.601424, -0.803434, 1.570796, 1.809992],accel_mss,speed_ms,0,blend_radius_m)
    movel([0.239196, -1.305333, -2.600340, -0.806716, 1.570796, 1.809992],accel_mss,speed_ms,0,blend_radius_m)
    movel([0.239196, -1.303147, -2.599252, -0.809991, 1.570796, 1.809992],accel_mss,speed_ms,0,blend_radius_m)
    movel([0.239196, -1.300972, -2.598160, -0.813257, 1.570796, 1.809992],accel_mss,speed_ms,0,blend_radius_m)
    movel([0.239196, -1.298808, -2.597065, -0.816516, 1.570796, 1.809992],accel_mss,speed_ms,0,blend_radius_m)
    movel([0.239196, -1.296656, -2.595967, -0.819766, 1.570796, 1.809992],accel_mss,speed_ms,0,blend_radius_m)
    movel([0.239196, -1.294515, -2.594865, -0.823009, 1.570796, 1.809992],accel_mss,speed_ms,0,blend_radius_m)
    movel([0.239196, -1.292386, -2.593759, -0.826244, 1.570796, 1.809992],accel_mss,speed_ms,0,blend_radius_m)
    movel([0.239196, -1.290267, -2.592650, -0.829471, 1.570796, 1.809992],accel_mss,speed_ms,0,blend_radius_m)
    movel([0.239196, -1.288161, -2.591538, -0.832691, 1.570796, 1.809992],accel_mss,speed_ms,0,blend_radius_m)
    movel([0.239196, -1.286065, -2.590422, -0.835902, 1.570796, 1.809992],accel_mss,speed_ms,0,blend_radius_m)
    # Splitting Linear movement in 10 (instruction 690: MoveL 559)
    movel([0.238194, -1.288552, -2.588940, -0.834896, 1.570796, 1.808991],accel_mss,speed_ms,0,blend_radius_m)
    movel([0.237198, -1.291031, -2.587457, -0.833902, 1.570796, 1.807995],accel_mss,speed_ms,0,blend_radius_m)
    movel([0.236208, -1.293499, -2.585971, -0.832919, 1.570796, 1.807004],accel_mss,speed_ms,0,blend_radius_m)
    movel([0.235222, -1.295959, -2.584484, -0.831947, 1.570796, 1.806018],accel_mss,speed_ms,0,blend_radius_m)
    movel([0.234242, -1.298409, -2.582994, -0.830986, 1.570796, 1.805038],accel_mss,speed_ms,0,blend_radius_m)
    movel([0.233266, -1.300850, -2.581503, -0.830036, 1.570796, 1.804063],accel_mss,speed_ms,0,blend_radius_m)
    movel([0.232296, -1.303282, -2.580009, -0.829098, 1.570796, 1.803093],accel_mss,speed_ms,0,blend_radius_m)
    movel([0.231331, -1.305705, -2.578514, -0.828170, 1.570796, 1.802127],accel_mss,speed_ms,0,blend_radius_m)
    movel([0.230371, -1.308118, -2.577017, -0.827253, 1.570796, 1.801167],accel_mss,speed_ms,0,blend_radius_m)
    movel([0.229416, -1.310523, -2.575518, -0.826347, 1.570796, 1.800212],accel_mss,speed_ms,0,blend_radius_m)
    # Splitting Linear movement in 12 (instruction 691: MoveL 560)
    movel([0.229416, -1.312591, -2.576608, -0.823190, 1.570796, 1.800212],accel_mss,speed_ms,0,blend_radius_m)
    movel([0.229416, -1.314669, -2.577694, -0.820026, 1.570796, 1.800212],accel_mss,speed_ms,0,blend_radius_m)
    movel([0.229416, -1.316758, -2.578776, -0.816855, 1.570796, 1.800212],accel_mss,speed_ms,0,blend_radius_m)
    movel([0.229416, -1.318858, -2.579855, -0.813676, 1.570796, 1.800212],accel_mss,speed_ms,0,blend_radius_m)
    movel([0.229416, -1.320968, -2.580931, -0.810490, 1.570796, 1.800212],accel_mss,speed_ms,0,blend_radius_m)
    movel([0.229416, -1.323089, -2.582003, -0.807297, 1.570796, 1.800212],accel_mss,speed_ms,0,blend_radius_m)
    movel([0.229416, -1.325220, -2.583072, -0.804097, 1.570796, 1.800212],accel_mss,speed_ms,0,blend_radius_m)
    movel([0.229416, -1.327363, -2.584137, -0.800890, 1.570796, 1.800212],accel_mss,speed_ms,0,blend_radius_m)
    movel([0.229416, -1.329516, -2.585198, -0.797675, 1.570796, 1.800212],accel_mss,speed_ms,0,blend_radius_m)
    movel([0.229416, -1.331680, -2.586256, -0.794453, 1.570796, 1.800212],accel_mss,speed_ms,0,blend_radius_m)
    movel([0.229416, -1.333855, -2.587310, -0.791224, 1.570796, 1.800212],accel_mss,speed_ms,0,blend_radius_m)
    movel([0.229416, -1.336041, -2.588360, -0.787988, 1.570796, 1.800212],accel_mss,speed_ms,0,blend_radius_m)
    speed_ms = 0.003
    # Splitting Linear movement in 6 (instruction 693: MoveL 561)
    movel([0.229416, -1.337687, -2.589146, -0.785556, 1.570796, 1.800212],accel_mss,speed_ms,0,blend_radius_m)
    movel([0.229416, -1.339339, -2.589929, -0.783121, 1.570796, 1.800212],accel_mss,speed_ms,0,blend_radius_m)
    movel([0.229416, -1.340998, -2.590710, -0.780681, 1.570796, 1.800212],accel_mss,speed_ms,0,blend_radius_m)
    movel([0.229416, -1.342663, -2.591490, -0.778237, 1.570796, 1.800212],accel_mss,speed_ms,0,blend_radius_m)
    movel([0.229416, -1.344334, -2.592267, -0.775789, 1.570796, 1.800212],accel_mss,speed_ms,0,blend_radius_m)
    movel([0.229416, -1.346011, -2.593042, -0.773337, 1.570796, 1.800212],accel_mss,speed_ms,0,blend_radius_m)
    speed_ms = 0.007
    movel([0.230067, -1.346402, -2.592784, -0.773203, 1.570796, 1.800863],accel_mss,speed_ms,0,blend_radius_m)
    movel([0.230044, -1.347066, -2.592347, -0.772976, 1.570796, 1.800841],accel_mss,speed_ms,0,blend_radius_m)
    movel([0.229686, -1.347676, -2.591944, -0.772769, 1.570796, 1.800483],accel_mss,speed_ms,0,blend_radius_m)
    movel([0.228540, -1.348320, -2.591519, -0.772550, 1.570796, 1.799337],accel_mss,speed_ms,0,blend_radius_m)
    movel([0.228452, -1.348326, -2.591515, -0.772548, 1.570796, 1.799248],accel_mss,speed_ms,0,blend_radius_m)
    movel([0.227802, -1.347934, -2.591774, -0.772681, 1.570796, 1.798598],accel_mss,speed_ms,0,blend_radius_m)
    movel([0.227822, -1.347274, -2.592210, -0.772906, 1.570796, 1.798618],accel_mss,speed_ms,0,blend_radius_m)
    movel([0.228179, -1.346662, -2.592613, -0.773114, 1.570796, 1.798975],accel_mss,speed_ms,0,blend_radius_m)
    movel([0.229327, -1.346016, -2.593038, -0.773335, 1.570796, 1.800124],accel_mss,speed_ms,0,blend_radius_m)
    movel([0.229416, -1.346011, -2.593042, -0.773337, 1.570796, 1.800212],accel_mss,speed_ms,0,blend_radius_m)
    speed_ms = 0.003
    movel([0.229416, -1.349383, -2.594586, -0.768420, 1.570796, 1.800212],accel_mss,speed_ms,0,blend_radius_m)
    speed_ms = 0.007
    movel([0.230067, -1.349773, -2.594327, -0.768288, 1.570796, 1.800863],accel_mss,speed_ms,0,blend_radius_m)
    movel([0.230044, -1.350435, -2.593889, -0.768065, 1.570796, 1.800841],accel_mss,speed_ms,0,blend_radius_m)
    movel([0.229686, -1.351045, -2.593485, -0.767859, 1.570796, 1.800483],accel_mss,speed_ms,0,blend_radius_m)
    movel([0.228540, -1.351687, -2.593059, -0.767643, 1.570796, 1.799337],accel_mss,speed_ms,0,blend_radius_m)
    movel([0.228452, -1.351692, -2.593055, -0.767642, 1.570796, 1.799248],accel_mss,speed_ms,0,blend_radius_m)
    movel([0.227802, -1.351301, -2.593315, -0.767773, 1.570796, 1.798598],accel_mss,speed_ms,0,blend_radius_m)
    movel([0.227822, -1.350643, -2.593751, -0.767995, 1.570796, 1.798618],accel_mss,speed_ms,0,blend_radius_m)
    movel([0.228179, -1.350033, -2.594155, -0.768200, 1.570796, 1.798975],accel_mss,speed_ms,0,blend_radius_m)
    movel([0.229327, -1.349388, -2.594582, -0.768419, 1.570796, 1.800124],accel_mss,speed_ms,0,blend_radius_m)
    movel([0.229416, -1.349383, -2.594586, -0.768420, 1.570796, 1.800212],accel_mss,speed_ms,0,blend_radius_m)
    speed_ms = 0.003
    # Splitting Linear movement in 8 (instruction 719: MoveL 583)
    movel([0.229416, -1.347694, -2.593815, -0.770881, 1.570796, 1.800212],accel_mss,speed_ms,0,blend_radius_m)
    movel([0.229416, -1.346011, -2.593042, -0.773337, 1.570796, 1.800212],accel_mss,speed_ms,0,blend_radius_m)
    movel([0.229416, -1.344334, -2.592267, -0.775789, 1.570796, 1.800212],accel_mss,speed_ms,0,blend_radius_m)
    movel([0.229416, -1.342663, -2.591490, -0.778237, 1.570796, 1.800212],accel_mss,speed_ms,0,blend_radius_m)
    movel([0.229416, -1.340998, -2.590710, -0.780681, 1.570796, 1.800212],accel_mss,speed_ms,0,blend_radius_m)
    movel([0.229416, -1.339339, -2.589929, -0.783121, 1.570796, 1.800212],accel_mss,speed_ms,0,blend_radius_m)
    movel([0.229416, -1.337687, -2.589146, -0.785556, 1.570796, 1.800212],accel_mss,speed_ms,0,blend_radius_m)
    movel([0.229416, -1.336041, -2.588360, -0.787988, 1.570796, 1.800212],accel_mss,speed_ms,0,blend_radius_m)
    speed_ms = 1.000
    # Splitting Linear movement in 12 (instruction 721: MoveL 584)
    movel([0.229416, -1.333855, -2.587310, -0.791224, 1.570796, 1.800212],accel_mss,speed_ms,0,blend_radius_m)
    movel([0.229416, -1.331680, -2.586256, -0.794453, 1.570796, 1.800212],accel_mss,speed_ms,0,blend_radius_m)
    movel([0.229416, -1.329516, -2.585198, -0.797675, 1.570796, 1.800212],accel_mss,speed_ms,0,blend_radius_m)
    movel([0.229416, -1.327363, -2.584137, -0.800890, 1.570796, 1.800212],accel_mss,speed_ms,0,blend_radius_m)
    movel([0.229416, -1.325220, -2.583072, -0.804097, 1.570796, 1.800212],accel_mss,speed_ms,0,blend_radius_m)
    movel([0.229416, -1.323089, -2.582003, -0.807297, 1.570796, 1.800212],accel_mss,speed_ms,0,blend_radius_m)
    movel([0.229416, -1.320968, -2.580931, -0.810490, 1.570796, 1.800212],accel_mss,speed_ms,0,blend_radius_m)
    movel([0.229416, -1.318858, -2.579855, -0.813676, 1.570796, 1.800212],accel_mss,speed_ms,0,blend_radius_m)
    movel([0.229416, -1.316758, -2.578776, -0.816855, 1.570796, 1.800212],accel_mss,speed_ms,0,blend_radius_m)
    movel([0.229416, -1.314669, -2.577694, -0.820026, 1.570796, 1.800212],accel_mss,speed_ms,0,blend_radius_m)
    movel([0.229416, -1.312591, -2.576608, -0.823190, 1.570796, 1.800212],accel_mss,speed_ms,0,blend_radius_m)
    movel([0.229416, -1.310523, -2.575518, -0.826347, 1.570796, 1.800212],accel_mss,speed_ms,0,blend_radius_m)
    # Splitting Linear movement in 8 (instruction 722: MoveL 585)
    movel([0.228744, -1.309145, -2.576378, -0.826866, 1.570796, 1.799540],accel_mss,speed_ms,0,blend_radius_m)
    movel([0.228069, -1.307766, -2.577236, -0.827387, 1.570796, 1.798866],accel_mss,speed_ms,0,blend_radius_m)
    movel([0.227392, -1.306385, -2.578093, -0.827911, 1.570796, 1.798189],accel_mss,speed_ms,0,blend_radius_m)
    movel([0.226713, -1.305003, -2.578948, -0.828438, 1.570796, 1.797509],accel_mss,speed_ms,0,blend_radius_m)
    movel([0.226031, -1.303620, -2.579801, -0.828968, 1.570796, 1.796828],accel_mss,speed_ms,0,blend_radius_m)
    movel([0.225347, -1.302236, -2.580653, -0.829501, 1.570796, 1.796144],accel_mss,speed_ms,0,blend_radius_m)
    movel([0.224661, -1.300850, -2.581502, -0.830036, 1.570796, 1.795457],accel_mss,speed_ms,0,blend_radius_m)
    movel([0.223972, -1.299464, -2.582351, -0.830575, 1.570796, 1.794768],accel_mss,speed_ms,0,blend_radius_m)
    # Splitting Linear movement in 14 (instruction 723: MoveL 586)
    movel([0.223972, -1.301246, -2.583295, -0.827848, 1.570796, 1.794768],accel_mss,speed_ms,0,blend_radius_m)
    movel([0.223972, -1.303037, -2.584237, -0.825115, 1.570796, 1.794768],accel_mss,speed_ms,0,blend_radius_m)
    movel([0.223972, -1.304836, -2.585176, -0.822377, 1.570796, 1.794768],accel_mss,speed_ms,0,blend_radius_m)
    movel([0.223972, -1.306643, -2.586113, -0.819634, 1.570796, 1.794768],accel_mss,speed_ms,0,blend_radius_m)
    movel([0.223972, -1.308457, -2.587047, -0.816885, 1.570796, 1.794768],accel_mss,speed_ms,0,blend_radius_m)
    movel([0.223972, -1.310280, -2.587978, -0.814130, 1.570796, 1.794768],accel_mss,speed_ms,0,blend_radius_m)
    movel([0.223972, -1.312111, -2.588907, -0.811371, 1.570796, 1.794768],accel_mss,speed_ms,0,blend_radius_m)
    movel([0.223972, -1.313950, -2.589833, -0.808605, 1.570796, 1.794768],accel_mss,speed_ms,0,blend_radius_m)
    movel([0.223972, -1.315798, -2.590757, -0.805834, 1.570796, 1.794768],accel_mss,speed_ms,0,blend_radius_m)
    movel([0.223972, -1.317653, -2.591678, -0.803058, 1.570796, 1.794768],accel_mss,speed_ms,0,blend_radius_m)
    movel([0.223972, -1.319516, -2.592597, -0.800276, 1.570796, 1.794768],accel_mss,speed_ms,0,blend_radius_m)
    movel([0.223972, -1.321388, -2.593512, -0.797488, 1.570796, 1.794768],accel_mss,speed_ms,0,blend_radius_m)
    movel([0.223972, -1.323268, -2.594426, -0.794695, 1.570796, 1.794768],accel_mss,speed_ms,0,blend_radius_m)
    movel([0.223972, -1.325156, -2.595336, -0.791897, 1.570796, 1.794768],accel_mss,speed_ms,0,blend_radius_m)
    speed_ms = 0.003
    # Splitting Linear movement in 6 (instruction 725: MoveL 587)
    movel([0.223972, -1.326815, -2.596131, -0.789444, 1.570796, 1.794768],accel_mss,speed_ms,0,blend_radius_m)
    movel([0.223972, -1.328480, -2.596923, -0.786986, 1.570796, 1.794768],accel_mss,speed_ms,0,blend_radius_m)
    movel([0.223972, -1.330151, -2.597713, -0.784525, 1.570796, 1.794768],accel_mss,speed_ms,0,blend_radius_m)
    movel([0.223972, -1.331828, -2.598502, -0.782059, 1.570796, 1.794768],accel_mss,speed_ms,0,blend_radius_m)
    movel([0.223972, -1.333512, -2.599288, -0.779589, 1.570796, 1.794768],accel_mss,speed_ms,0,blend_radius_m)
    movel([0.223972, -1.335203, -2.600072, -0.777115, 1.570796, 1.794768],accel_mss,speed_ms,0,blend_radius_m)
    speed_ms = 0.007
    # Splitting Linear movement in 6 (instruction 727: MoveL 588)
    movel([0.224549, -1.333478, -2.601179, -0.777732, 1.570796, 1.795345],accel_mss,speed_ms,0,blend_radius_m)
    movel([0.225129, -1.331749, -2.602285, -0.778355, 1.570796, 1.795925],accel_mss,speed_ms,0,blend_radius_m)
    movel([0.225710, -1.330015, -2.603390, -0.778984, 1.570796, 1.796507],accel_mss,speed_ms,0,blend_radius_m)
    movel([0.226295, -1.328276, -2.604494, -0.779619, 1.570796, 1.797091],accel_mss,speed_ms,0,blend_radius_m)
    movel([0.226881, -1.326532, -2.605597, -0.780260, 1.570796, 1.797677],accel_mss,speed_ms,0,blend_radius_m)
    movel([0.227470, -1.324783, -2.606699, -0.780907, 1.570796, 1.798266],accel_mss,speed_ms,0,blend_radius_m)
    # Splitting Linear movement in 14 (instruction 728: MoveL 589)
    movel([0.229841, -1.324535, -2.606855, -0.780999, 1.570796, 1.800637],accel_mss,speed_ms,0,blend_radius_m)
    movel([0.232211, -1.324293, -2.607007, -0.781089, 1.570796, 1.803007],accel_mss,speed_ms,0,blend_radius_m)
    movel([0.234580, -1.324056, -2.607156, -0.781177, 1.570796, 1.805376],accel_mss,speed_ms,0,blend_radius_m)
    movel([0.236947, -1.323824, -2.607302, -0.781263, 1.570796, 1.807744],accel_mss,speed_ms,0,blend_radius_m)
    movel([0.239314, -1.323597, -2.607445, -0.781348, 1.570796, 1.810110],accel_mss,speed_ms,0,blend_radius_m)
    movel([0.241679, -1.323375, -2.607584, -0.781431, 1.570796, 1.812475],accel_mss,speed_ms,0,blend_radius_m)
    movel([0.244042, -1.323158, -2.607719, -0.781511, 1.570796, 1.814838],accel_mss,speed_ms,0,blend_radius_m)
    movel([0.246404, -1.322947, -2.607852, -0.781590, 1.570796, 1.817200],accel_mss,speed_ms,0,blend_radius_m)
    movel([0.248765, -1.322741, -2.607981, -0.781667, 1.570796, 1.819561],accel_mss,speed_ms,0,blend_radius_m)
    movel([0.251124, -1.322540, -2.608107, -0.781742, 1.570796, 1.821920],accel_mss,speed_ms,0,blend_radius_m)
    movel([0.253482, -1.322344, -2.608230, -0.781816, 1.570796, 1.824278],accel_mss,speed_ms,0,blend_radius_m)
    movel([0.255838, -1.322153, -2.608349, -0.781887, 1.570796, 1.826634],accel_mss,speed_ms,0,blend_radius_m)
    movel([0.258192, -1.321968, -2.608465, -0.781956, 1.570796, 1.828989],accel_mss,speed_ms,0,blend_radius_m)
    movel([0.260546, -1.321788, -2.608577, -0.782024, 1.570796, 1.831342],accel_mss,speed_ms,0,blend_radius_m)
    # Splitting Linear movement in 6 (instruction 729: MoveL 590)
    movel([0.260240, -1.323525, -2.607489, -0.781374, 1.570796, 1.831037],accel_mss,speed_ms,0,blend_radius_m)
    movel([0.259936, -1.325258, -2.606400, -0.780731, 1.570796, 1.830733],accel_mss,speed_ms,0,blend_radius_m)
    movel([0.259633, -1.326987, -2.605310, -0.780093, 1.570796, 1.830430],accel_mss,speed_ms,0,blend_radius_m)
    movel([0.259332, -1.328710, -2.604218, -0.779460, 1.570796, 1.830128],accel_mss,speed_ms,0,blend_radius_m)
    movel([0.259031, -1.330429, -2.603126, -0.778834, 1.570796, 1.829828],accel_mss,speed_ms,0,blend_radius_m)
    movel([0.258732, -1.332144, -2.602033, -0.778213, 1.570796, 1.829529],accel_mss,speed_ms,0,blend_radius_m)
    movel([0.256576, -1.332302, -2.601932, -0.778156, 1.570796, 1.827372],accel_mss,speed_ms,0,blend_radius_m)
    # Splitting Linear movement in 14 (instruction 731: MoveL 592)
    movel([0.254256, -1.332476, -2.601820, -0.778093, 1.570796, 1.825052],accel_mss,speed_ms,0,blend_radius_m)
    movel([0.251935, -1.332656, -2.601705, -0.778028, 1.570796, 1.822731],accel_mss,speed_ms,0,blend_radius_m)
    movel([0.249612, -1.332840, -2.601587, -0.777961, 1.570796, 1.820409],accel_mss,speed_ms,0,blend_radius_m)
    movel([0.247288, -1.333030, -2.601466, -0.777893, 1.570796, 1.818084],accel_mss,speed_ms,0,blend_radius_m)
    movel([0.244962, -1.333225, -2.601341, -0.777823, 1.570796, 1.815759],accel_mss,speed_ms,0,blend_radius_m)
    movel([0.242635, -1.333425, -2.601213, -0.777751, 1.570796, 1.813432],accel_mss,speed_ms,0,blend_radius_m)
    movel([0.240307, -1.333629, -2.601082, -0.777678, 1.570796, 1.811103],accel_mss,speed_ms,0,blend_radius_m)
    movel([0.237977, -1.333839, -2.600947, -0.777602, 1.570796, 1.808774],accel_mss,speed_ms,0,blend_radius_m)
    movel([0.235646, -1.334054, -2.600810, -0.777525, 1.570796, 1.806442],accel_mss,speed_ms,0,blend_radius_m)
    movel([0.233314, -1.334274, -2.600669, -0.777447, 1.570796, 1.804110],accel_mss,speed_ms,0,blend_radius_m)
    movel([0.230980, -1.334498, -2.600524, -0.777366, 1.570796, 1.801776],accel_mss,speed_ms,0,blend_radius_m)
    movel([0.228645, -1.334728, -2.600377, -0.777284, 1.570796, 1.799442],accel_mss,speed_ms,0,blend_radius_m)
    movel([0.226309, -1.334963, -2.600226, -0.777200, 1.570796, 1.797105],accel_mss,speed_ms,0,blend_radius_m)
    movel([0.223972, -1.335203, -2.600072, -0.777115, 1.570796, 1.794768],accel_mss,speed_ms,0,blend_radius_m)
    speed_ms = 0.003
    movel([0.223972, -1.338602, -2.601634, -0.772153, 1.570796, 1.794768],accel_mss,speed_ms,0,blend_radius_m)
    speed_ms = 0.007
    # Splitting Linear movement in 6 (instruction 735: MoveL 594)
    movel([0.224549, -1.336882, -2.602743, -0.772764, 1.570796, 1.795345],accel_mss,speed_ms,0,blend_radius_m)
    movel([0.225129, -1.335157, -2.603852, -0.773380, 1.570796, 1.795925],accel_mss,speed_ms,0,blend_radius_m)
    movel([0.225710, -1.333427, -2.604960, -0.774002, 1.570796, 1.796507],accel_mss,speed_ms,0,blend_radius_m)
    movel([0.226295, -1.331692, -2.606067, -0.774629, 1.570796, 1.797091],accel_mss,speed_ms,0,blend_radius_m)
    movel([0.226881, -1.329952, -2.607173, -0.775263, 1.570796, 1.797677],accel_mss,speed_ms,0,blend_radius_m)
    movel([0.227470, -1.328208, -2.608279, -0.775903, 1.570796, 1.798266],accel_mss,speed_ms,0,blend_radius_m)
    # Splitting Linear movement in 14 (instruction 736: MoveL 595)
    movel([0.229841, -1.327961, -2.608435, -0.775994, 1.570796, 1.800637],accel_mss,speed_ms,0,blend_radius_m)
    movel([0.232211, -1.327719, -2.608587, -0.776083, 1.570796, 1.803007],accel_mss,speed_ms,0,blend_radius_m)
    movel([0.234580, -1.327482, -2.608737, -0.776170, 1.570796, 1.805376],accel_mss,speed_ms,0,blend_radius_m)
    movel([0.236947, -1.327251, -2.608883, -0.776255, 1.570796, 1.807744],accel_mss,speed_ms,0,blend_radius_m)
    movel([0.239314, -1.327024, -2.609026, -0.776339, 1.570796, 1.810110],accel_mss,speed_ms,0,blend_radius_m)
    movel([0.241679, -1.326803, -2.609165, -0.776421, 1.570796, 1.812475],accel_mss,speed_ms,0,blend_radius_m)
    movel([0.244042, -1.326587, -2.609302, -0.776501, 1.570796, 1.814838],accel_mss,speed_ms,0,blend_radius_m)
    movel([0.246404, -1.326376, -2.609434, -0.776579, 1.570796, 1.817200],accel_mss,speed_ms,0,blend_radius_m)
    movel([0.248765, -1.326170, -2.609564, -0.776655, 1.570796, 1.819561],accel_mss,speed_ms,0,blend_radius_m)
    movel([0.251124, -1.325970, -2.609690, -0.776729, 1.570796, 1.821920],accel_mss,speed_ms,0,blend_radius_m)
    movel([0.253482, -1.325774, -2.609813, -0.776802, 1.570796, 1.824278],accel_mss,speed_ms,0,blend_radius_m)
    movel([0.255838, -1.325584, -2.609933, -0.776872, 1.570796, 1.826634],accel_mss,speed_ms,0,blend_radius_m)
    movel([0.258192, -1.325399, -2.610049, -0.776941, 1.570796, 1.828989],accel_mss,speed_ms,0,blend_radius_m)
    movel([0.260546, -1.325220, -2.610162, -0.777008, 1.570796, 1.831342],accel_mss,speed_ms,0,blend_radius_m)
    # Splitting Linear movement in 6 (instruction 737: MoveL 596)
    movel([0.260240, -1.326953, -2.609071, -0.776365, 1.570796, 1.831037],accel_mss,speed_ms,0,blend_radius_m)
    movel([0.259936, -1.328682, -2.607979, -0.775728, 1.570796, 1.830733],accel_mss,speed_ms,0,blend_radius_m)
    movel([0.259633, -1.330406, -2.606885, -0.775097, 1.570796, 1.830430],accel_mss,speed_ms,0,blend_radius_m)
    movel([0.259332, -1.332126, -2.605791, -0.774472, 1.570796, 1.830128],accel_mss,speed_ms,0,blend_radius_m)
    movel([0.259031, -1.333841, -2.604696, -0.773853, 1.570796, 1.829828],accel_mss,speed_ms,0,blend_radius_m)
    movel([0.258732, -1.335551, -2.603600, -0.773239, 1.570796, 1.829529],accel_mss,speed_ms,0,blend_radius_m)
    movel([0.256576, -1.335708, -2.603498, -0.773182, 1.570796, 1.827372],accel_mss,speed_ms,0,blend_radius_m)
    # Splitting Linear movement in 14 (instruction 739: MoveL 598)
    movel([0.254256, -1.335882, -2.603387, -0.773120, 1.570796, 1.825052],accel_mss,speed_ms,0,blend_radius_m)
    movel([0.251935, -1.336061, -2.603271, -0.773056, 1.570796, 1.822731],accel_mss,speed_ms,0,blend_radius_m)
    movel([0.249612, -1.336246, -2.603153, -0.772990, 1.570796, 1.820409],accel_mss,speed_ms,0,blend_radius_m)
    movel([0.247288, -1.336435, -2.603031, -0.772923, 1.570796, 1.818084],accel_mss,speed_ms,0,blend_radius_m)
    movel([0.244962, -1.336629, -2.602906, -0.772854, 1.570796, 1.815759],accel_mss,speed_ms,0,blend_radius_m)
    movel([0.242635, -1.336828, -2.602778, -0.772783, 1.570796, 1.813432],accel_mss,speed_ms,0,blend_radius_m)
    movel([0.240307, -1.337033, -2.602646, -0.772710, 1.570796, 1.811103],accel_mss,speed_ms,0,blend_radius_m)
    movel([0.237977, -1.337242, -2.602512, -0.772635, 1.570796, 1.808774],accel_mss,speed_ms,0,blend_radius_m)
    movel([0.235646, -1.337456, -2.602373, -0.772559, 1.570796, 1.806442],accel_mss,speed_ms,0,blend_radius_m)
    movel([0.233314, -1.337675, -2.602232, -0.772482, 1.570796, 1.804110],accel_mss,speed_ms,0,blend_radius_m)
    movel([0.230980, -1.337900, -2.602087, -0.772402, 1.570796, 1.801776],accel_mss,speed_ms,0,blend_radius_m)
    movel([0.228645, -1.338129, -2.601939, -0.772321, 1.570796, 1.799442],accel_mss,speed_ms,0,blend_radius_m)
    movel([0.226309, -1.338363, -2.601788, -0.772238, 1.570796, 1.797105],accel_mss,speed_ms,0,blend_radius_m)
    movel([0.223972, -1.338602, -2.601634, -0.772153, 1.570796, 1.794768],accel_mss,speed_ms,0,blend_radius_m)
    speed_ms = 0.003
    # Splitting Linear movement in 6 (instruction 741: MoveL 599)
    movel([0.223972, -1.336333, -2.600593, -0.775463, 1.570796, 1.794768],accel_mss,speed_ms,0,blend_radius_m)
    movel([0.223972, -1.334075, -2.599549, -0.778765, 1.570796, 1.794768],accel_mss,speed_ms,0,blend_radius_m)
    movel([0.223972, -1.331828, -2.598502, -0.782059, 1.570796, 1.794768],accel_mss,speed_ms,0,blend_radius_m)
    movel([0.223972, -1.329593, -2.597450, -0.785346, 1.570796, 1.794768],accel_mss,speed_ms,0,blend_radius_m)
    movel([0.223972, -1.327369, -2.596395, -0.788625, 1.570796, 1.794768],accel_mss,speed_ms,0,blend_radius_m)
    movel([0.223972, -1.325156, -2.595336, -0.791897, 1.570796, 1.794768],accel_mss,speed_ms,0,blend_radius_m)
    speed_ms = 1.000
    # Splitting Linear movement in 14 (instruction 743: MoveL 600)
    movel([0.223972, -1.323268, -2.594426, -0.794695, 1.570796, 1.794768],accel_mss,speed_ms,0,blend_radius_m)
    movel([0.223972, -1.321388, -2.593512, -0.797488, 1.570796, 1.794768],accel_mss,speed_ms,0,blend_radius_m)
    movel([0.223972, -1.319516, -2.592597, -0.800276, 1.570796, 1.794768],accel_mss,speed_ms,0,blend_radius_m)
    movel([0.223972, -1.317653, -2.591678, -0.803058, 1.570796, 1.794768],accel_mss,speed_ms,0,blend_radius_m)
    movel([0.223972, -1.315798, -2.590757, -0.805834, 1.570796, 1.794768],accel_mss,speed_ms,0,blend_radius_m)
    movel([0.223972, -1.313950, -2.589833, -0.808605, 1.570796, 1.794768],accel_mss,speed_ms,0,blend_radius_m)
    movel([0.223972, -1.312111, -2.588907, -0.811371, 1.570796, 1.794768],accel_mss,speed_ms,0,blend_radius_m)
    movel([0.223972, -1.310280, -2.587978, -0.814130, 1.570796, 1.794768],accel_mss,speed_ms,0,blend_radius_m)
    movel([0.223972, -1.308457, -2.587047, -0.816885, 1.570796, 1.794768],accel_mss,speed_ms,0,blend_radius_m)
    movel([0.223972, -1.306643, -2.586113, -0.819634, 1.570796, 1.794768],accel_mss,speed_ms,0,blend_radius_m)
    movel([0.223972, -1.304836, -2.585176, -0.822377, 1.570796, 1.794768],accel_mss,speed_ms,0,blend_radius_m)
    movel([0.223972, -1.303037, -2.584237, -0.825115, 1.570796, 1.794768],accel_mss,speed_ms,0,blend_radius_m)
    movel([0.223972, -1.301246, -2.583295, -0.827848, 1.570796, 1.794768],accel_mss,speed_ms,0,blend_radius_m)
    movel([0.223972, -1.299464, -2.582351, -0.830575, 1.570796, 1.794768],accel_mss,speed_ms,0,blend_radius_m)
    # Splitting Linear movement in 8 (instruction 744: MoveL 601)
    movel([0.225908, -1.297655, -2.583453, -0.831281, 1.570796, 1.796704],accel_mss,speed_ms,0,blend_radius_m)
    movel([0.227851, -1.295843, -2.584554, -0.831992, 1.570796, 1.798647],accel_mss,speed_ms,0,blend_radius_m)
    movel([0.229800, -1.294027, -2.585652, -0.832709, 1.570796, 1.800596],accel_mss,speed_ms,0,blend_radius_m)
    movel([0.231756, -1.292208, -2.586749, -0.833432, 1.570796, 1.802552],accel_mss,speed_ms,0,blend_radius_m)
    movel([0.233718, -1.290384, -2.587844, -0.834160, 1.570796, 1.804514],accel_mss,speed_ms,0,blend_radius_m)
    movel([0.235687, -1.288557, -2.588937, -0.834894, 1.570796, 1.806483],accel_mss,speed_ms,0,blend_radius_m)
    movel([0.237662, -1.286726, -2.590028, -0.835634, 1.570796, 1.808458],accel_mss,speed_ms,0,blend_radius_m)
    movel([0.239644, -1.284892, -2.591118, -0.836379, 1.570796, 1.810440],accel_mss,speed_ms,0,blend_radius_m)
    # Splitting Linear movement in 14 (instruction 745: MoveL 602)
    movel([0.239644, -1.286689, -2.592075, -0.833625, 1.570796, 1.810440],accel_mss,speed_ms,0,blend_radius_m)
    movel([0.239644, -1.288494, -2.593031, -0.830865, 1.570796, 1.810440],accel_mss,speed_ms,0,blend_radius_m)
    movel([0.239644, -1.290307, -2.593983, -0.828099, 1.570796, 1.810440],accel_mss,speed_ms,0,blend_radius_m)
    movel([0.239644, -1.292128, -2.594934, -0.825327, 1.570796, 1.810440],accel_mss,speed_ms,0,blend_radius_m)
    movel([0.239644, -1.293958, -2.595881, -0.822549, 1.570796, 1.810440],accel_mss,speed_ms,0,blend_radius_m)
    movel([0.239644, -1.295797, -2.596826, -0.819766, 1.570796, 1.810440],accel_mss,speed_ms,0,blend_radius_m)
    movel([0.239644, -1.297643, -2.597769, -0.816977, 1.570796, 1.810440],accel_mss,speed_ms,0,blend_radius_m)
    movel([0.239644, -1.299498, -2.598709, -0.814182, 1.570796, 1.810440],accel_mss,speed_ms,0,blend_radius_m)
    movel([0.239644, -1.301362, -2.599646, -0.811381, 1.570796, 1.810440],accel_mss,speed_ms,0,blend_radius_m)
    movel([0.239644, -1.303234, -2.600581, -0.808575, 1.570796, 1.810440],accel_mss,speed_ms,0,blend_radius_m)
    movel([0.239644, -1.305114, -2.601513, -0.805762, 1.570796, 1.810440],accel_mss,speed_ms,0,blend_radius_m)
    movel([0.239644, -1.307003, -2.602442, -0.802944, 1.570796, 1.810440],accel_mss,speed_ms,0,blend_radius_m)
    movel([0.239644, -1.308900, -2.603369, -0.800120, 1.570796, 1.810440],accel_mss,speed_ms,0,blend_radius_m)
    movel([0.239644, -1.310806, -2.604293, -0.797291, 1.570796, 1.810440],accel_mss,speed_ms,0,blend_radius_m)
    speed_ms = 0.003
    # Splitting Linear movement in 6 (instruction 747: MoveL 603)
    movel([0.239644, -1.312480, -2.605099, -0.794810, 1.570796, 1.810440],accel_mss,speed_ms,0,blend_radius_m)
    movel([0.239644, -1.314161, -2.605904, -0.792324, 1.570796, 1.810440],accel_mss,speed_ms,0,blend_radius_m)
    movel([0.239644, -1.315848, -2.606706, -0.789835, 1.570796, 1.810440],accel_mss,speed_ms,0,blend_radius_m)
    movel([0.239644, -1.317542, -2.607506, -0.787340, 1.570796, 1.810440],accel_mss,speed_ms,0,blend_radius_m)
    movel([0.239644, -1.319243, -2.608304, -0.784842, 1.570796, 1.810440],accel_mss,speed_ms,0,blend_radius_m)
    movel([0.239644, -1.320950, -2.609100, -0.782338, 1.570796, 1.810440],accel_mss,speed_ms,0,blend_radius_m)
    speed_ms = 0.007
    # Splitting Linear movement in 4 (instruction 749: MoveC 604)
    movel([0.238696, -1.320373, -2.609460, -0.782556, 1.570796, 1.809493],accel_mss,speed_ms,0,blend_radius_m)
    movel([0.237747, -1.319797, -2.609819, -0.782773, 1.570796, 1.808543],accel_mss,speed_ms,0,blend_radius_m)
    movel([0.236795, -1.319222, -2.610176, -0.782990, 1.570796, 1.807592],accel_mss,speed_ms,0,blend_radius_m)
    movel([0.235843, -1.318648, -2.610533, -0.783208, 1.570796, 1.806639],accel_mss,speed_ms,0,blend_radius_m)
    movel([0.236031, -1.314861, -2.612875, -0.784653, 1.570796, 1.806827],accel_mss,speed_ms,0,blend_radius_m)
    movel([0.238881, -1.310495, -2.615551, -0.786343, 1.570796, 1.809677],accel_mss,speed_ms,0,blend_radius_m)
    # Splitting Linear movement in 4 (instruction 752: MoveC 607)
    movel([0.240350, -1.309736, -2.616014, -0.786639, 1.570796, 1.811146],accel_mss,speed_ms,0,blend_radius_m)
    movel([0.241821, -1.308976, -2.616476, -0.786937, 1.570796, 1.812618],accel_mss,speed_ms,0,blend_radius_m)
    movel([0.243294, -1.308217, -2.616937, -0.787234, 1.570796, 1.814091],accel_mss,speed_ms,0,blend_radius_m)
    movel([0.244769, -1.307458, -2.617398, -0.787533, 1.570796, 1.815565],accel_mss,speed_ms,0,blend_radius_m)
    movel([0.245186, -1.307433, -2.617413, -0.787543, 1.570796, 1.815983],accel_mss,speed_ms,0,blend_radius_m)
    # Splitting Linear movement in 4 (instruction 754: MoveC 609)
    movel([0.246142, -1.308023, -2.617055, -0.787311, 1.570796, 1.816938],accel_mss,speed_ms,0,blend_radius_m)
    movel([0.247095, -1.308613, -2.616697, -0.787079, 1.570796, 1.817891],accel_mss,speed_ms,0,blend_radius_m)
    movel([0.248046, -1.309205, -2.616337, -0.786847, 1.570796, 1.818843],accel_mss,speed_ms,0,blend_radius_m)
    movel([0.248996, -1.309797, -2.615977, -0.786615, 1.570796, 1.819793],accel_mss,speed_ms,0,blend_radius_m)
    movel([0.248752, -1.313632, -2.613631, -0.785126, 1.570796, 1.819549],accel_mss,speed_ms,0,blend_radius_m)
    movel([0.245872, -1.317968, -2.610955, -0.783466, 1.570796, 1.816669],accel_mss,speed_ms,0,blend_radius_m)
    # Splitting Linear movement in 4 (instruction 757: MoveC 612)
    movel([0.244416, -1.318707, -2.610497, -0.783186, 1.570796, 1.815212],accel_mss,speed_ms,0,blend_radius_m)
    movel([0.242961, -1.319445, -2.610038, -0.782906, 1.570796, 1.813758],accel_mss,speed_ms,0,blend_radius_m)
    movel([0.241508, -1.320184, -2.609578, -0.782627, 1.570796, 1.812304],accel_mss,speed_ms,0,blend_radius_m)
    movel([0.240056, -1.320924, -2.609117, -0.782348, 1.570796, 1.810853],accel_mss,speed_ms,0,blend_radius_m)
    movel([0.239644, -1.320950, -2.609100, -0.782338, 1.570796, 1.810440],accel_mss,speed_ms,0,blend_radius_m)
    speed_ms = 0.003
    movel([0.239644, -1.324384, -2.610686, -0.777319, 1.570796, 1.810440],accel_mss,speed_ms,0,blend_radius_m)
    speed_ms = 0.007
    # Splitting Linear movement in 4 (instruction 762: MoveC 615)
    movel([0.238696, -1.323809, -2.611047, -0.777534, 1.570796, 1.809493],accel_mss,speed_ms,0,blend_radius_m)
    movel([0.237747, -1.323234, -2.611407, -0.777748, 1.570796, 1.808543],accel_mss,speed_ms,0,blend_radius_m)
    movel([0.236795, -1.322660, -2.611765, -0.777964, 1.570796, 1.807592],accel_mss,speed_ms,0,blend_radius_m)
    movel([0.235843, -1.322088, -2.612123, -0.778179, 1.570796, 1.806639],accel_mss,speed_ms,0,blend_radius_m)
    movel([0.236031, -1.318310, -2.614471, -0.779609, 1.570796, 1.806827],accel_mss,speed_ms,0,blend_radius_m)
    movel([0.238881, -1.313954, -2.617154, -0.781281, 1.570796, 1.809677],accel_mss,speed_ms,0,blend_radius_m)
    # Splitting Linear movement in 4 (instruction 765: MoveC 618)
    movel([0.240350, -1.313196, -2.617619, -0.781574, 1.570796, 1.811146],accel_mss,speed_ms,0,blend_radius_m)
    movel([0.241821, -1.312438, -2.618082, -0.781869, 1.570796, 1.812618],accel_mss,speed_ms,0,blend_radius_m)
    movel([0.243294, -1.311681, -2.618545, -0.782163, 1.570796, 1.814091],accel_mss,speed_ms,0,blend_radius_m)
    movel([0.244769, -1.310924, -2.619006, -0.782459, 1.570796, 1.815565],accel_mss,speed_ms,0,blend_radius_m)
    movel([0.245186, -1.310899, -2.619022, -0.782469, 1.570796, 1.815983],accel_mss,speed_ms,0,blend_radius_m)
    # Splitting Linear movement in 4 (instruction 767: MoveC 620)
    movel([0.246142, -1.311487, -2.618663, -0.782239, 1.570796, 1.816938],accel_mss,speed_ms,0,blend_radius_m)
    movel([0.247095, -1.312076, -2.618304, -0.782009, 1.570796, 1.817891],accel_mss,speed_ms,0,blend_radius_m)
    movel([0.248046, -1.312666, -2.617943, -0.781780, 1.570796, 1.818843],accel_mss,speed_ms,0,blend_radius_m)
    movel([0.248996, -1.313257, -2.617581, -0.781551, 1.570796, 1.819793],accel_mss,speed_ms,0,blend_radius_m)
    movel([0.248752, -1.317083, -2.615229, -0.780077, 1.570796, 1.819549],accel_mss,speed_ms,0,blend_radius_m)
    movel([0.245872, -1.321409, -2.612546, -0.778434, 1.570796, 1.816669],accel_mss,speed_ms,0,blend_radius_m)
    # Splitting Linear movement in 4 (instruction 770: MoveC 623)
    movel([0.244416, -1.322146, -2.612086, -0.778157, 1.570796, 1.815212],accel_mss,speed_ms,0,blend_radius_m)
    movel([0.242961, -1.322883, -2.611626, -0.777880, 1.570796, 1.813758],accel_mss,speed_ms,0,blend_radius_m)
    movel([0.241508, -1.323620, -2.611165, -0.777604, 1.570796, 1.812304],accel_mss,speed_ms,0,blend_radius_m)
    movel([0.240056, -1.324358, -2.610703, -0.777329, 1.570796, 1.810853],accel_mss,speed_ms,0,blend_radius_m)
    movel([0.239644, -1.324384, -2.610686, -0.777319, 1.570796, 1.810440],accel_mss,speed_ms,0,blend_radius_m)
    speed_ms = 0.003
    # Splitting Linear movement in 6 (instruction 773: MoveL 625)
    movel([0.239644, -1.322092, -2.609630, -0.780667, 1.570796, 1.810440],accel_mss,speed_ms,0,blend_radius_m)
    movel([0.239644, -1.319811, -2.608570, -0.784008, 1.570796, 1.810440],accel_mss,speed_ms,0,blend_radius_m)
    movel([0.239644, -1.317542, -2.607506, -0.787340, 1.570796, 1.810440],accel_mss,speed_ms,0,blend_radius_m)
    movel([0.239644, -1.315285, -2.606439, -0.790665, 1.570796, 1.810440],accel_mss,speed_ms,0,blend_radius_m)
    movel([0.239644, -1.313040, -2.605368, -0.793982, 1.570796, 1.810440],accel_mss,speed_ms,0,blend_radius_m)
    movel([0.239644, -1.310806, -2.604293, -0.797291, 1.570796, 1.810440],accel_mss,speed_ms,0,blend_radius_m)
    speed_ms = 1.000
    # Splitting Linear movement in 14 (instruction 775: MoveL 626)
    movel([0.239644, -1.308900, -2.603369, -0.800120, 1.570796, 1.810440],accel_mss,speed_ms,0,blend_radius_m)
    movel([0.239644, -1.307003, -2.602442, -0.802944, 1.570796, 1.810440],accel_mss,speed_ms,0,blend_radius_m)
    movel([0.239644, -1.305114, -2.601513, -0.805762, 1.570796, 1.810440],accel_mss,speed_ms,0,blend_radius_m)
    movel([0.239644, -1.303234, -2.600581, -0.808575, 1.570796, 1.810440],accel_mss,speed_ms,0,blend_radius_m)
    movel([0.239644, -1.301362, -2.599646, -0.811381, 1.570796, 1.810440],accel_mss,speed_ms,0,blend_radius_m)
    movel([0.239644, -1.299498, -2.598709, -0.814182, 1.570796, 1.810440],accel_mss,speed_ms,0,blend_radius_m)
    movel([0.239644, -1.297643, -2.597769, -0.816977, 1.570796, 1.810440],accel_mss,speed_ms,0,blend_radius_m)
    movel([0.239644, -1.295797, -2.596826, -0.819766, 1.570796, 1.810440],accel_mss,speed_ms,0,blend_radius_m)
    movel([0.239644, -1.293958, -2.595881, -0.822549, 1.570796, 1.810440],accel_mss,speed_ms,0,blend_radius_m)
    movel([0.239644, -1.292128, -2.594934, -0.825327, 1.570796, 1.810440],accel_mss,speed_ms,0,blend_radius_m)
    movel([0.239644, -1.290307, -2.593983, -0.828099, 1.570796, 1.810440],accel_mss,speed_ms,0,blend_radius_m)
    movel([0.239644, -1.288494, -2.593031, -0.830865, 1.570796, 1.810440],accel_mss,speed_ms,0,blend_radius_m)
    movel([0.239644, -1.286689, -2.592075, -0.833625, 1.570796, 1.810440],accel_mss,speed_ms,0,blend_radius_m)
    movel([0.239644, -1.284892, -2.591118, -0.836379, 1.570796, 1.810440],accel_mss,speed_ms,0,blend_radius_m)
    # Splitting Linear movement in 8 (instruction 776: MoveL 627)
    movel([0.241722, -1.285490, -2.590763, -0.836136, 1.570796, 1.812518],accel_mss,speed_ms,0,blend_radius_m)
    movel([0.243795, -1.286092, -2.590405, -0.835891, 1.570796, 1.814591],accel_mss,speed_ms,0,blend_radius_m)
    movel([0.245863, -1.286701, -2.590044, -0.835645, 1.570796, 1.816659],accel_mss,speed_ms,0,blend_radius_m)
    movel([0.247926, -1.287314, -2.589679, -0.835396, 1.570796, 1.818722],accel_mss,speed_ms,0,blend_radius_m)
    movel([0.249984, -1.287932, -2.589310, -0.835147, 1.570796, 1.820780],accel_mss,speed_ms,0,blend_radius_m)
    movel([0.252037, -1.288556, -2.588938, -0.834895, 1.570796, 1.822834],accel_mss,speed_ms,0,blend_radius_m)
    movel([0.254086, -1.289184, -2.588563, -0.834642, 1.570796, 1.824882],accel_mss,speed_ms,0,blend_radius_m)
    movel([0.256129, -1.289818, -2.588184, -0.834388, 1.570796, 1.826925],accel_mss,speed_ms,0,blend_radius_m)
    # Splitting Linear movement in 14 (instruction 777: MoveL 628)
    movel([0.256129, -1.291610, -2.589137, -0.831642, 1.570796, 1.826925],accel_mss,speed_ms,0,blend_radius_m)
    movel([0.256129, -1.293410, -2.590088, -0.828891, 1.570796, 1.826925],accel_mss,speed_ms,0,blend_radius_m)
    movel([0.256129, -1.295218, -2.591036, -0.826135, 1.570796, 1.826925],accel_mss,speed_ms,0,blend_radius_m)
    movel([0.256129, -1.297035, -2.591981, -0.823372, 1.570796, 1.826925],accel_mss,speed_ms,0,blend_radius_m)
    movel([0.256129, -1.298860, -2.592924, -0.820604, 1.570796, 1.826925],accel_mss,speed_ms,0,blend_radius_m)
    movel([0.256129, -1.300693, -2.593865, -0.817831, 1.570796, 1.826925],accel_mss,speed_ms,0,blend_radius_m)
    movel([0.256129, -1.302535, -2.594803, -0.815052, 1.570796, 1.826925],accel_mss,speed_ms,0,blend_radius_m)
    movel([0.256129, -1.304384, -2.595738, -0.812266, 1.570796, 1.826925],accel_mss,speed_ms,0,blend_radius_m)
    movel([0.256129, -1.306242, -2.596671, -0.809476, 1.570796, 1.826925],accel_mss,speed_ms,0,blend_radius_m)
    movel([0.256129, -1.308109, -2.597601, -0.806679, 1.570796, 1.826925],accel_mss,speed_ms,0,blend_radius_m)
    movel([0.256129, -1.309983, -2.598528, -0.803877, 1.570796, 1.826925],accel_mss,speed_ms,0,blend_radius_m)
    movel([0.256129, -1.311866, -2.599453, -0.801069, 1.570796, 1.826925],accel_mss,speed_ms,0,blend_radius_m)
    movel([0.256129, -1.313758, -2.600375, -0.798256, 1.570796, 1.826925],accel_mss,speed_ms,0,blend_radius_m)
    movel([0.256129, -1.315658, -2.601295, -0.795437, 1.570796, 1.826925],accel_mss,speed_ms,0,blend_radius_m)
    speed_ms = 0.003
    # Splitting Linear movement in 6 (instruction 779: MoveL 629)
    movel([0.256129, -1.317327, -2.602097, -0.792965, 1.570796, 1.826925],accel_mss,speed_ms,0,blend_radius_m)
    movel([0.256129, -1.319003, -2.602897, -0.790489, 1.570796, 1.826925],accel_mss,speed_ms,0,blend_radius_m)
    movel([0.256129, -1.320685, -2.603696, -0.788009, 1.570796, 1.826925],accel_mss,speed_ms,0,blend_radius_m)
    movel([0.256129, -1.322373, -2.604492, -0.785524, 1.570796, 1.826925],accel_mss,speed_ms,0,blend_radius_m)
    movel([0.256129, -1.324068, -2.605286, -0.783035, 1.570796, 1.826925],accel_mss,speed_ms,0,blend_radius_m)
    movel([0.256129, -1.325770, -2.606078, -0.780541, 1.570796, 1.826925],accel_mss,speed_ms,0,blend_radius_m)
    speed_ms = 0.007
    movel([0.260342, -1.325055, -2.606528, -0.780806, 1.570796, 1.831138],accel_mss,speed_ms,0,blend_radius_m)
    movel([0.264790, -1.325457, -2.606275, -0.780657, 1.570796, 1.835586],accel_mss,speed_ms,0,blend_radius_m)
    movel([0.265876, -1.325805, -2.606056, -0.780529, 1.570796, 1.836672],accel_mss,speed_ms,0,blend_radius_m)
    movel([0.268499, -1.327269, -2.605131, -0.779989, 1.570796, 1.839295],accel_mss,speed_ms,0,blend_radius_m)
    # Splitting Linear movement in 4 (instruction 785: MoveC 634)
    movel([0.269255, -1.328312, -2.604471, -0.779606, 1.570796, 1.840051],accel_mss,speed_ms,0,blend_radius_m)
    movel([0.270008, -1.329356, -2.603809, -0.779225, 1.570796, 1.840804],accel_mss,speed_ms,0,blend_radius_m)
    movel([0.270759, -1.330399, -2.603145, -0.778845, 1.570796, 1.841556],accel_mss,speed_ms,0,blend_radius_m)
    movel([0.271508, -1.331442, -2.602481, -0.778466, 1.570796, 1.842305],accel_mss,speed_ms,0,blend_radius_m)
    movel([0.272098, -1.333771, -2.600991, -0.777627, 1.570796, 1.842895],accel_mss,speed_ms,0,blend_radius_m)
    movel([0.272381, -1.337895, -2.598335, -0.776158, 1.570796, 1.843178],accel_mss,speed_ms,0,blend_radius_m)
    movel([0.272339, -1.339425, -2.597344, -0.775620, 1.570796, 1.843136],accel_mss,speed_ms,0,blend_radius_m)
    movel([0.272201, -1.342072, -2.595622, -0.774695, 1.570796, 1.842998],accel_mss,speed_ms,0,blend_radius_m)
    movel([0.272106, -1.343766, -2.594515, -0.774108, 1.570796, 1.842902],accel_mss,speed_ms,0,blend_radius_m)
    movel([0.272065, -1.344712, -2.593895, -0.773782, 1.570796, 1.842861],accel_mss,speed_ms,0,blend_radius_m)
    # Splitting Linear movement in 6 (instruction 792: MoveC 641)
    movel([0.272141, -1.346232, -2.592896, -0.773261, 1.570796, 1.842937],accel_mss,speed_ms,0,blend_radius_m)
    movel([0.272216, -1.347749, -2.591896, -0.772744, 1.570796, 1.843012],accel_mss,speed_ms,0,blend_radius_m)
    movel([0.272291, -1.349262, -2.590895, -0.772231, 1.570796, 1.843087],accel_mss,speed_ms,0,blend_radius_m)
    movel([0.272366, -1.350773, -2.589893, -0.771723, 1.570796, 1.843162],accel_mss,speed_ms,0,blend_radius_m)
    movel([0.272440, -1.352280, -2.588890, -0.771219, 1.570796, 1.843236],accel_mss,speed_ms,0,blend_radius_m)
    movel([0.272514, -1.353784, -2.587886, -0.770719, 1.570796, 1.843311],accel_mss,speed_ms,0,blend_radius_m)
    movel([0.273160, -1.357307, -2.585522, -0.769560, 1.570796, 1.843956],accel_mss,speed_ms,0,blend_radius_m)
    # Splitting Linear movement in 4 (instruction 794: MoveC 643)
    movel([0.272894, -1.356292, -2.586205, -0.769892, 1.570796, 1.843690],accel_mss,speed_ms,0,blend_radius_m)
    movel([0.272627, -1.355275, -2.586888, -0.770226, 1.570796, 1.843423],accel_mss,speed_ms,0,blend_radius_m)
    movel([0.272359, -1.354257, -2.587570, -0.770562, 1.570796, 1.843156],accel_mss,speed_ms,0,blend_radius_m)
    movel([0.272091, -1.353238, -2.588251, -0.770900, 1.570796, 1.842887],accel_mss,speed_ms,0,blend_radius_m)
    # Splitting Linear movement in 4 (instruction 795: MoveC 644)
    movel([0.271849, -1.351214, -2.589600, -0.771575, 1.570796, 1.842645],accel_mss,speed_ms,0,blend_radius_m)
    movel([0.271606, -1.349184, -2.590947, -0.772258, 1.570796, 1.842402],accel_mss,speed_ms,0,blend_radius_m)
    movel([0.271362, -1.347149, -2.592292, -0.772948, 1.570796, 1.842158],accel_mss,speed_ms,0,blend_radius_m)
    movel([0.271116, -1.345108, -2.593635, -0.773646, 1.570796, 1.841912],accel_mss,speed_ms,0,blend_radius_m)
    movel([0.271096, -1.344472, -2.594052, -0.773865, 1.570796, 1.841892],accel_mss,speed_ms,0,blend_radius_m)
    movel([0.271079, -1.343653, -2.594589, -0.774147, 1.570796, 1.841876],accel_mss,speed_ms,0,blend_radius_m)
    movel([0.271052, -1.341931, -2.595714, -0.774744, 1.570796, 1.841849],accel_mss,speed_ms,0,blend_radius_m)
    movel([0.271006, -1.339826, -2.597084, -0.775479, 1.570796, 1.841802],accel_mss,speed_ms,0,blend_radius_m)
    movel([0.270944, -1.338529, -2.597925, -0.775935, 1.570796, 1.841740],accel_mss,speed_ms,0,blend_radius_m)
    movel([0.270355, -1.334647, -2.600429, -0.777313, 1.570796, 1.841152],accel_mss,speed_ms,0,blend_radius_m)
    movel([0.269673, -1.332742, -2.601650, -0.777997, 1.570796, 1.840469],accel_mss,speed_ms,0,blend_radius_m)
    # Splitting Linear movement in 4 (instruction 803: MoveC 652)
    movel([0.268816, -1.331831, -2.602232, -0.778326, 1.570796, 1.839613],accel_mss,speed_ms,0,blend_radius_m)
    movel([0.267958, -1.330921, -2.602813, -0.778655, 1.570796, 1.838754],accel_mss,speed_ms,0,blend_radius_m)
    movel([0.267097, -1.330012, -2.603392, -0.778985, 1.570796, 1.837893],accel_mss,speed_ms,0,blend_radius_m)
    movel([0.266234, -1.329103, -2.603969, -0.779317, 1.570796, 1.837030],accel_mss,speed_ms,0,blend_radius_m)
    movel([0.264214, -1.328278, -2.604492, -0.779618, 1.570796, 1.835010],accel_mss,speed_ms,0,blend_radius_m)
    movel([0.263237, -1.328057, -2.604632, -0.779699, 1.570796, 1.834033],accel_mss,speed_ms,0,blend_radius_m)
    movel([0.259425, -1.327975, -2.604684, -0.779729, 1.570796, 1.830222],accel_mss,speed_ms,0,blend_radius_m)
    movel([0.257397, -1.328329, -2.604460, -0.779600, 1.570796, 1.828194],accel_mss,speed_ms,0,blend_radius_m)
    movel([0.255697, -1.328815, -2.604152, -0.779422, 1.570796, 1.826493],accel_mss,speed_ms,0,blend_radius_m)
    movel([0.256129, -1.325770, -2.606078, -0.780541, 1.570796, 1.826925],accel_mss,speed_ms,0,blend_radius_m)
    speed_ms = 0.003
    movel([0.256129, -1.329192, -2.607656, -0.775541, 1.570796, 1.826925],accel_mss,speed_ms,0,blend_radius_m)
    speed_ms = 0.007
    movel([0.260342, -1.328479, -2.608107, -0.775803, 1.570796, 1.831138],accel_mss,speed_ms,0,blend_radius_m)
    movel([0.264790, -1.328881, -2.607853, -0.775656, 1.570796, 1.835586],accel_mss,speed_ms,0,blend_radius_m)
    movel([0.265876, -1.329227, -2.607634, -0.775529, 1.570796, 1.836672],accel_mss,speed_ms,0,blend_radius_m)
    movel([0.268499, -1.330688, -2.606707, -0.774995, 1.570796, 1.839295],accel_mss,speed_ms,0,blend_radius_m)
    # Splitting Linear movement in 4 (instruction 817: MoveC 664)
    movel([0.269255, -1.331729, -2.606044, -0.774616, 1.570796, 1.840051],accel_mss,speed_ms,0,blend_radius_m)
    movel([0.270008, -1.332769, -2.605380, -0.774239, 1.570796, 1.840804],accel_mss,speed_ms,0,blend_radius_m)
    movel([0.270759, -1.333810, -2.604715, -0.773864, 1.570796, 1.841556],accel_mss,speed_ms,0,blend_radius_m)
    movel([0.271508, -1.334850, -2.604049, -0.773490, 1.570796, 1.842305],accel_mss,speed_ms,0,blend_radius_m)
    movel([0.272098, -1.337174, -2.602555, -0.772660, 1.570796, 1.842895],accel_mss,speed_ms,0,blend_radius_m)
    movel([0.272381, -1.341288, -2.599893, -0.771208, 1.570796, 1.843178],accel_mss,speed_ms,0,blend_radius_m)
    movel([0.272339, -1.342814, -2.598899, -0.770676, 1.570796, 1.843136],accel_mss,speed_ms,0,blend_radius_m)
    movel([0.272201, -1.345454, -2.597173, -0.769762, 1.570796, 1.842998],accel_mss,speed_ms,0,blend_radius_m)
    movel([0.272106, -1.347145, -2.596062, -0.769182, 1.570796, 1.842902],accel_mss,speed_ms,0,blend_radius_m)
    movel([0.272065, -1.348088, -2.595441, -0.768860, 1.570796, 1.842861],accel_mss,speed_ms,0,blend_radius_m)
    # Splitting Linear movement in 6 (instruction 824: MoveC 671)
    movel([0.272141, -1.349604, -2.594439, -0.768345, 1.570796, 1.842937],accel_mss,speed_ms,0,blend_radius_m)
    movel([0.272216, -1.351117, -2.593437, -0.767835, 1.570796, 1.843012],accel_mss,speed_ms,0,blend_radius_m)
    movel([0.272291, -1.352626, -2.592434, -0.767329, 1.570796, 1.843087],accel_mss,speed_ms,0,blend_radius_m)
    movel([0.272366, -1.354133, -2.591429, -0.766827, 1.570796, 1.843162],accel_mss,speed_ms,0,blend_radius_m)
    movel([0.272440, -1.355636, -2.590424, -0.766329, 1.570796, 1.843236],accel_mss,speed_ms,0,blend_radius_m)
    movel([0.272514, -1.357136, -2.589417, -0.765835, 1.570796, 1.843311],accel_mss,speed_ms,0,blend_radius_m)
    movel([0.273160, -1.360651, -2.587047, -0.764691, 1.570796, 1.843956],accel_mss,speed_ms,0,blend_radius_m)
    # Splitting Linear movement in 4 (instruction 826: MoveC 673)
    movel([0.272894, -1.359638, -2.587732, -0.765019, 1.570796, 1.843690],accel_mss,speed_ms,0,blend_radius_m)
    movel([0.272627, -1.358624, -2.588416, -0.765349, 1.570796, 1.843423],accel_mss,speed_ms,0,blend_radius_m)
    movel([0.272359, -1.357609, -2.589100, -0.765681, 1.570796, 1.843156],accel_mss,speed_ms,0,blend_radius_m)
    movel([0.272091, -1.356592, -2.589783, -0.766014, 1.570796, 1.842887],accel_mss,speed_ms,0,blend_radius_m)
    # Splitting Linear movement in 4 (instruction 827: MoveC 674)
    movel([0.271849, -1.354573, -2.591135, -0.766681, 1.570796, 1.842645],accel_mss,speed_ms,0,blend_radius_m)
    movel([0.271606, -1.352548, -2.592486, -0.767355, 1.570796, 1.842402],accel_mss,speed_ms,0,blend_radius_m)
    movel([0.271362, -1.350518, -2.593834, -0.768037, 1.570796, 1.842158],accel_mss,speed_ms,0,blend_radius_m)
    movel([0.271116, -1.348483, -2.595180, -0.768726, 1.570796, 1.841912],accel_mss,speed_ms,0,blend_radius_m)
    movel([0.271096, -1.347848, -2.595599, -0.768942, 1.570796, 1.841892],accel_mss,speed_ms,0,blend_radius_m)
    movel([0.271079, -1.347031, -2.596137, -0.769221, 1.570796, 1.841876],accel_mss,speed_ms,0,blend_radius_m)
    movel([0.271052, -1.345314, -2.597265, -0.769811, 1.570796, 1.841849],accel_mss,speed_ms,0,blend_radius_m)
    movel([0.271006, -1.343214, -2.598639, -0.770537, 1.570796, 1.841802],accel_mss,speed_ms,0,blend_radius_m)
    movel([0.270944, -1.341920, -2.599482, -0.770987, 1.570796, 1.841740],accel_mss,speed_ms,0,blend_radius_m)
    movel([0.270355, -1.338048, -2.601992, -0.772350, 1.570796, 1.841152],accel_mss,speed_ms,0,blend_radius_m)
    movel([0.269673, -1.336147, -2.603216, -0.773026, 1.570796, 1.840469],accel_mss,speed_ms,0,blend_radius_m)
    # Splitting Linear movement in 4 (instruction 835: MoveC 682)
    movel([0.268816, -1.335239, -2.603800, -0.773350, 1.570796, 1.839613],accel_mss,speed_ms,0,blend_radius_m)
    movel([0.267958, -1.334331, -2.604382, -0.773676, 1.570796, 1.838754],accel_mss,speed_ms,0,blend_radius_m)
    movel([0.267097, -1.333424, -2.604962, -0.774003, 1.570796, 1.837893],accel_mss,speed_ms,0,blend_radius_m)
    movel([0.266234, -1.332517, -2.605542, -0.774330, 1.570796, 1.837030],accel_mss,speed_ms,0,blend_radius_m)
    movel([0.264214, -1.331695, -2.606066, -0.774628, 1.570796, 1.835010],accel_mss,speed_ms,0,blend_radius_m)
    movel([0.263237, -1.331474, -2.606206, -0.774709, 1.570796, 1.834033],accel_mss,speed_ms,0,blend_radius_m)
    movel([0.259425, -1.331392, -2.606258, -0.774738, 1.570796, 1.830222],accel_mss,speed_ms,0,blend_radius_m)
    movel([0.257397, -1.331745, -2.606033, -0.774610, 1.570796, 1.828194],accel_mss,speed_ms,0,blend_radius_m)
    movel([0.255697, -1.332231, -2.605724, -0.774434, 1.570796, 1.826493],accel_mss,speed_ms,0,blend_radius_m)
    movel([0.256129, -1.329192, -2.607656, -0.775541, 1.570796, 1.826925],accel_mss,speed_ms,0,blend_radius_m)
    speed_ms = 0.003
    # Splitting Linear movement in 8 (instruction 843: MoveL 689)
    movel([0.256129, -1.327478, -2.606868, -0.778044, 1.570796, 1.826925],accel_mss,speed_ms,0,blend_radius_m)
    movel([0.256129, -1.325770, -2.606078, -0.780541, 1.570796, 1.826925],accel_mss,speed_ms,0,blend_radius_m)
    movel([0.256129, -1.324068, -2.605286, -0.783035, 1.570796, 1.826925],accel_mss,speed_ms,0,blend_radius_m)
    movel([0.256129, -1.322373, -2.604492, -0.785524, 1.570796, 1.826925],accel_mss,speed_ms,0,blend_radius_m)
    movel([0.256129, -1.320685, -2.603696, -0.788009, 1.570796, 1.826925],accel_mss,speed_ms,0,blend_radius_m)
    movel([0.256129, -1.319003, -2.602897, -0.790489, 1.570796, 1.826925],accel_mss,speed_ms,0,blend_radius_m)
    movel([0.256129, -1.317327, -2.602097, -0.792965, 1.570796, 1.826925],accel_mss,speed_ms,0,blend_radius_m)
    movel([0.256129, -1.315658, -2.601295, -0.795437, 1.570796, 1.826925],accel_mss,speed_ms,0,blend_radius_m)
    speed_ms = 1.000
    # Splitting Linear movement in 14 (instruction 845: MoveL 690)
    movel([0.256129, -1.313758, -2.600375, -0.798256, 1.570796, 1.826925],accel_mss,speed_ms,0,blend_radius_m)
    movel([0.256129, -1.311866, -2.599453, -0.801069, 1.570796, 1.826925],accel_mss,speed_ms,0,blend_radius_m)
    movel([0.256129, -1.309983, -2.598528, -0.803877, 1.570796, 1.826925],accel_mss,speed_ms,0,blend_radius_m)
    movel([0.256129, -1.308109, -2.597601, -0.806679, 1.570796, 1.826925],accel_mss,speed_ms,0,blend_radius_m)
    movel([0.256129, -1.306242, -2.596671, -0.809476, 1.570796, 1.826925],accel_mss,speed_ms,0,blend_radius_m)
    movel([0.256129, -1.304384, -2.595738, -0.812266, 1.570796, 1.826925],accel_mss,speed_ms,0,blend_radius_m)
    movel([0.256129, -1.302535, -2.594803, -0.815052, 1.570796, 1.826925],accel_mss,speed_ms,0,blend_radius_m)
    movel([0.256129, -1.300693, -2.593865, -0.817831, 1.570796, 1.826925],accel_mss,speed_ms,0,blend_radius_m)
    movel([0.256129, -1.298860, -2.592924, -0.820604, 1.570796, 1.826925],accel_mss,speed_ms,0,blend_radius_m)
    movel([0.256129, -1.297035, -2.591981, -0.823372, 1.570796, 1.826925],accel_mss,speed_ms,0,blend_radius_m)
    movel([0.256129, -1.295218, -2.591036, -0.826135, 1.570796, 1.826925],accel_mss,speed_ms,0,blend_radius_m)
    movel([0.256129, -1.293410, -2.590088, -0.828891, 1.570796, 1.826925],accel_mss,speed_ms,0,blend_radius_m)
    movel([0.256129, -1.291610, -2.589137, -0.831642, 1.570796, 1.826925],accel_mss,speed_ms,0,blend_radius_m)
    movel([0.256129, -1.289818, -2.588184, -0.834388, 1.570796, 1.826925],accel_mss,speed_ms,0,blend_radius_m)
    # Splitting Linear movement in 18 (instruction 846: MoveL 691)
    movel([0.257016, -1.291454, -2.587202, -0.833733, 1.570796, 1.827812],accel_mss,speed_ms,0,blend_radius_m)
    movel([0.257899, -1.293089, -2.586218, -0.833081, 1.570796, 1.828696],accel_mss,speed_ms,0,blend_radius_m)
    movel([0.258779, -1.294723, -2.585232, -0.832434, 1.570796, 1.829576],accel_mss,speed_ms,0,blend_radius_m)
    movel([0.259655, -1.296355, -2.584243, -0.831791, 1.570796, 1.830452],accel_mss,speed_ms,0,blend_radius_m)
    movel([0.260528, -1.297986, -2.583252, -0.831151, 1.570796, 1.831324],accel_mss,speed_ms,0,blend_radius_m)
    movel([0.261396, -1.299615, -2.582258, -0.830516, 1.570796, 1.832193],accel_mss,speed_ms,0,blend_radius_m)
    movel([0.262261, -1.301243, -2.581262, -0.829884, 1.570796, 1.833058],accel_mss,speed_ms,0,blend_radius_m)
    movel([0.263123, -1.302869, -2.580263, -0.829257, 1.570796, 1.833919],accel_mss,speed_ms,0,blend_radius_m)
    movel([0.263981, -1.304494, -2.579262, -0.828633, 1.570796, 1.834777],accel_mss,speed_ms,0,blend_radius_m)
    movel([0.264835, -1.306117, -2.578259, -0.828013, 1.570796, 1.835631],accel_mss,speed_ms,0,blend_radius_m)
    movel([0.265686, -1.307739, -2.577253, -0.827397, 1.570796, 1.836482],accel_mss,speed_ms,0,blend_radius_m)
    movel([0.266533, -1.309360, -2.576244, -0.826785, 1.570796, 1.837329],accel_mss,speed_ms,0,blend_radius_m)
    movel([0.267376, -1.310979, -2.575233, -0.826177, 1.570796, 1.838173],accel_mss,speed_ms,0,blend_radius_m)
    movel([0.268217, -1.312596, -2.574220, -0.825573, 1.570796, 1.839013],accel_mss,speed_ms,0,blend_radius_m)
    movel([0.269053, -1.314212, -2.573205, -0.824972, 1.570796, 1.839850],accel_mss,speed_ms,0,blend_radius_m)
    movel([0.269886, -1.315827, -2.572187, -0.824376, 1.570796, 1.840683],accel_mss,speed_ms,0,blend_radius_m)
    movel([0.270716, -1.317440, -2.571166, -0.823783, 1.570796, 1.841512],accel_mss,speed_ms,0,blend_radius_m)
    movel([0.271542, -1.319051, -2.570143, -0.823195, 1.570796, 1.842339],accel_mss,speed_ms,0,blend_radius_m)
    # Splitting Linear movement in 12 (instruction 847: MoveL 692)
    movel([0.271542, -1.321108, -2.571224, -0.820057, 1.570796, 1.842339],accel_mss,speed_ms,0,blend_radius_m)
    movel([0.271542, -1.323176, -2.572301, -0.816913, 1.570796, 1.842339],accel_mss,speed_ms,0,blend_radius_m)
    movel([0.271542, -1.325254, -2.573374, -0.813761, 1.570796, 1.842339],accel_mss,speed_ms,0,blend_radius_m)
    movel([0.271542, -1.327342, -2.574444, -0.810603, 1.570796, 1.842339],accel_mss,speed_ms,0,blend_radius_m)
    movel([0.271542, -1.329441, -2.575510, -0.807437, 1.570796, 1.842339],accel_mss,speed_ms,0,blend_radius_m)
    movel([0.271542, -1.331551, -2.576573, -0.804265, 1.570796, 1.842339],accel_mss,speed_ms,0,blend_radius_m)
    movel([0.271542, -1.333671, -2.577633, -0.801086, 1.570796, 1.842339],accel_mss,speed_ms,0,blend_radius_m)
    movel([0.271542, -1.335801, -2.578688, -0.797899, 1.570796, 1.842339],accel_mss,speed_ms,0,blend_radius_m)
    movel([0.271542, -1.337942, -2.579740, -0.794706, 1.570796, 1.842339],accel_mss,speed_ms,0,blend_radius_m)
    movel([0.271542, -1.340094, -2.580789, -0.791506, 1.570796, 1.842339],accel_mss,speed_ms,0,blend_radius_m)
    movel([0.271542, -1.342256, -2.581834, -0.788299, 1.570796, 1.842339],accel_mss,speed_ms,0,blend_radius_m)
    movel([0.271542, -1.344429, -2.582875, -0.785085, 1.570796, 1.842339],accel_mss,speed_ms,0,blend_radius_m)
    speed_ms = 0.003
    # Splitting Linear movement in 6 (instruction 849: MoveL 693)
    movel([0.271542, -1.346066, -2.583654, -0.782670, 1.570796, 1.842339],accel_mss,speed_ms,0,blend_radius_m)
    movel([0.271542, -1.347708, -2.584430, -0.780251, 1.570796, 1.842339],accel_mss,speed_ms,0,blend_radius_m)
    movel([0.271542, -1.349357, -2.585205, -0.777828, 1.570796, 1.842339],accel_mss,speed_ms,0,blend_radius_m)
    movel([0.271542, -1.351011, -2.585977, -0.775401, 1.570796, 1.842339],accel_mss,speed_ms,0,blend_radius_m)
    movel([0.271542, -1.352672, -2.586747, -0.772970, 1.570796, 1.842339],accel_mss,speed_ms,0,blend_radius_m)
    movel([0.271542, -1.354338, -2.587515, -0.770535, 1.570796, 1.842339],accel_mss,speed_ms,0,blend_radius_m)
    speed_ms = 0.007
    # Splitting Linear movement in 4 (instruction 851: MoveC 694)
    movel([0.272981, -1.354008, -2.587737, -0.770645, 1.570796, 1.843777],accel_mss,speed_ms,0,blend_radius_m)
    movel([0.274420, -1.353678, -2.587957, -0.770754, 1.570796, 1.845216],accel_mss,speed_ms,0,blend_radius_m)
    movel([0.275859, -1.353351, -2.588176, -0.770863, 1.570796, 1.846655],accel_mss,speed_ms,0,blend_radius_m)
    movel([0.277298, -1.353024, -2.588394, -0.770971, 1.570796, 1.848094],accel_mss,speed_ms,0,blend_radius_m)
    movel([0.277754, -1.353301, -2.588209, -0.770879, 1.570796, 1.848550],accel_mss,speed_ms,0,blend_radius_m)
    movel([0.278765, -1.354879, -2.587153, -0.770357, 1.570796, 1.849561],accel_mss,speed_ms,0,blend_radius_m)
    movel([0.278077, -1.358523, -2.584702, -0.769164, 1.570796, 1.848873],accel_mss,speed_ms,0,blend_radius_m)
    movel([0.276774, -1.360340, -2.583473, -0.768576, 1.570796, 1.847570],accel_mss,speed_ms,0,blend_radius_m)
    movel([0.275491, -1.361514, -2.582676, -0.768199, 1.570796, 1.846287],accel_mss,speed_ms,0,blend_radius_m)
    # Splitting Linear movement in 4 (instruction 857: MoveC 700)
    movel([0.274066, -1.361834, -2.582459, -0.768096, 1.570796, 1.844863],accel_mss,speed_ms,0,blend_radius_m)
    movel([0.272642, -1.362154, -2.582241, -0.767994, 1.570796, 1.843439],accel_mss,speed_ms,0,blend_radius_m)
    movel([0.271218, -1.362476, -2.582022, -0.767891, 1.570796, 1.842014],accel_mss,speed_ms,0,blend_radius_m)
    movel([0.269794, -1.362800, -2.581801, -0.767788, 1.570796, 1.840591],accel_mss,speed_ms,0,blend_radius_m)
    movel([0.269337, -1.362530, -2.581985, -0.767874, 1.570796, 1.840133],accel_mss,speed_ms,0,blend_radius_m)
    movel([0.268313, -1.360982, -2.583037, -0.768370, 1.570796, 1.839110],accel_mss,speed_ms,0,blend_radius_m)
    movel([0.268959, -1.357363, -2.585484, -0.769542, 1.570796, 1.839755],accel_mss,speed_ms,0,blend_radius_m)
    movel([0.270254, -1.355533, -2.586715, -0.770141, 1.570796, 1.841050],accel_mss,speed_ms,0,blend_radius_m)
    movel([0.271542, -1.354338, -2.587515, -0.770535, 1.570796, 1.842339],accel_mss,speed_ms,0,blend_radius_m)
    speed_ms = 0.003
    movel([0.271542, -1.357690, -2.589045, -0.765654, 1.570796, 1.842339],accel_mss,speed_ms,0,blend_radius_m)
    speed_ms = 0.007
    # Splitting Linear movement in 4 (instruction 866: MoveC 707)
    movel([0.272981, -1.357360, -2.589267, -0.765762, 1.570796, 1.843777],accel_mss,speed_ms,0,blend_radius_m)
